		station.xCycleEnable:=FALSE;	
		station.xDone:=TRUE;
		station.xRunningOffProhibit := FALSE ;//运行中信号Off禁止
	1000://XY轴回参考点
				fbXAxisMove.xMoveAuto[1]:=TRUE;
				fbYAxisMove.xMoveAuto[1]:=TRUE;
			IF	fbxAxisMove.xMoveInPos[1] AND 
				fbYAxisMove.xMoveInPos[1] THEN
					station.iStepAuto:= 0;
			END_IF		
{region "清料程序"}
  1010://开始请料
		 //写入数据
			arMainlineFixtureData[arCurFixtureNumStation[5]].xMaterialOnOff:=FALSE;
			arMainlineFixtureData[arCurFixtureNumStation[6]].xMaterialOnOff:=FALSE;
			arMainlineFixtureData[arCurFixtureNumStation[7]].xMaterialOnOff:=FALSE;
			arMainlineFixtureData[arCurFixtureNumStation[8]].xMaterialOnOff:=FALSE;
			arMainlineFixtureData[arCurFixtureNumStation[9]].xMaterialOnOff:=FALSE;		
			arMainlineFixtureData[arCurFixtureNumStation[5]].stProduct.xLidChecking_NOK:=TRUE;
			arMainlineFixtureData[arCurFixtureNumStation[5]].stProduct.xLidChecking_OK:=FALSE;	
			arMainlineFixtureData[arCurFixtureNumStation[6]].stProduct.xLidChecking_NOK:=TRUE;
			arMainlineFixtureData[arCurFixtureNumStation[6]].stProduct.xLidChecking_OK:=FALSE;	
			arMainlineFixtureData[arCurFixtureNumStation[7]].stProduct.xLidChecking_NOK:=TRUE;
			arMainlineFixtureData[arCurFixtureNumStation[7]].stProduct.xLidChecking_OK:=FALSE;	
			arMainlineFixtureData[arCurFixtureNumStation[8]].stProduct.xLidChecking_NOK:=TRUE;
			arMainlineFixtureData[arCurFixtureNumStation[8]].stProduct.xLidChecking_OK:=FALSE;	
			arMainlineFixtureData[arCurFixtureNumStation[9]].stProduct.xLidChecking_NOK:=TRUE;
			arMainlineFixtureData[arCurFixtureNumStation[9]].stProduct.xLidChecking_OK:=FALSE;	
			arMainlineFixtureData[arCurFixtureNumStation[5]].stProduct.xEmptying:=TRUE;
			arMainlineFixtureData[arCurFixtureNumStation[6]].stProduct.xEmptying:=TRUE;
			arMainlineFixtureData[arCurFixtureNumStation[7]].stProduct.xEmptying:=TRUE;
			arMainlineFixtureData[arCurFixtureNumStation[8]].stProduct.xEmptying:=TRUE;
			arMainlineFixtureData[arCurFixtureNumStation[9]].stProduct.xEmptying:=TRUE;		
			station.iStepAuto:=1020;
 1020://XY轴回参考点
				fbXAxisMove.xMoveAuto[1]:=TRUE;
				fbYAxisMove.xMoveAuto[1]:=TRUE;
			IF	fbxAxisMove.xMoveInPos[1] AND 
				fbYAxisMove.xMoveInPos[1] THEN
					station.iStepAuto:= 1100;
			END_IF			
 1100://清料完成
			station.xEmptying:=FALSE;
			station.xEmptyDone:=TRUE;
			station.iStepAuto:=0;
{endregion}			
			
			
			
			
			
		
	ELSE
		;	
END_CASE



END_IF
END_ACTION

ACTION FlowInit:
IF NOT station.xIniting THEN
  station.iStepInit:=0;    
ELSE
//--------------------------------------------初始化步序----------------------------------
CASE station.iStepInit OF	
 0://  
 
  	IF station.xIniting THEN	
  	  station.iStepInit:=10;	
  	END_IF	
10://复位数据
		MEMSET(ADR(arCameraResult),0,SIZEOF(arCameraResult));
		MEMSET(ADR(arCameraResultHmi),0,SIZEOF(arCameraResultHmi));
		FOR i:=2 TO 17 BY 1 DO
			fbCamera[i].xlInit:=TRUE;
			fbCamera[i].xlTrigger:=FALSE;
		END_FOR
		FOR i:=1 TO gc_ModuleProNo BY 1 DO
					MEMSET(ADR(tsModuleProcess[i]),0,SIZEOF(tsModuleProcess[i]));
				END_FOR
		station.iStepInit :=20;
	 
20://伺服上电
  	fbXAxisMove.xPowerInit := TRUE ;
	 fbYAxisMove.xPowerInit := TRUE ;
	 fbZAxisMove.xPowerInit := TRUE ;
	IF fbXAxisMove.xPowerOn AND   fbYAxisMove.xPowerOn AND  fbZAxisMove.xPowerOn THEN 
    	station.iStepInit:=30;	
	END_IF
30://Z轴伺服上升
		fbZAxisMove.xMoveAuto[1]:=TRUE;
		IF fbZAxisMove.xMoveInPos[1]   THEN
			station.iStepInit:=40;	
		END_IF
40://XY轴回参考位置
		fbXAxisMove.xMoveAuto[1]:=TRUE;
		fbYAxisMove.xMoveAuto[1]:=TRUE;
		IF fbXAxisMove.xMoveInPos[1]  AND   fbYAxisMove.xMoveInPos[1]  THEN
			station.iStepInit:=50;	
		END_IF
50://水平调整气缸回原位
				fbHOZAdjustCyl_1.xinit:=TRUE;
        fbHOZAdjustCyl_2.xinit:=TRUE;
        fbHOZAdjustCyl_3.xinit:=true;
       	fbHOZAdjustCyl_4.xinit:=TRUE;
        fbHOZAdjustCyl_5.xinit:=true;
      	fbHOZAdjustCyl_6.xinit:=TRUE;
        fbHOZAdjustCyl_7.xinit:=true;
      	 fbHOZAdjustCyl_8.xinit:=TRUE;
	IF  fbHOZAdjustCyl_1.xHP_Delay AND 
			fbHOZAdjustCyl_2.xHP_Delay AND
			fbHOZAdjustCyl_3.xHP_Delay AND
			fbHOZAdjustCyl_4.xHP_Delay AND 
			fbHOZAdjustCyl_5.xHP_Delay AND 
			fbHOZAdjustCyl_6.xHP_Delay AND
			fbHOZAdjustCyl_7.xHP_Delay AND
			fbHOZAdjustCyl_8.xHP_Delay THEN
		station.iStepInit:=60;	
	END_IF

60://
	station.iStepInit:=100;

100://	
    station.iStepInit:=999;	
999://初始化完成	
	station.iStepInit:=0;
	station.xInitDone:=TRUE;  
END_CASE
END_IF
END_ACTION

ACTION General:
{region "清除过程记录"}
CASE bClearProcessStep OF
	0:	
		IF	 S08_MainLine.xClearProcessStatus THEN
			FOR i:=1 TO gc_ModuleProNo BY 1 DO
				MEMSET(ADR(tsModuleProcess[i]),0,SIZEOF(tsModuleProcess[i]));
			END_FOR
			bClearProcessStep:=10;
		END_IF
	10:
		xClearModuleProcessDone:=TRUE;
		bClearProcessStep:=20;
	20:
		IF NOT S08_MainLine.xClearProcessStatus THEN
			xClearModuleProcessDone:=FALSE;
			bClearProcessStep:=30;
		END_IF
	30:  
			bClearProcessStep:=0;
	
END_CASE
{endregion}

{region "HMI中操作bCounter计数"}
IF station.xSingleRunning THEN
bCounter:=bS03Counter;
END_IF
{endregion}
END_ACTION

ACTION ILC:

//---------------------------------------------------工站可执行-------------------------------------------------------
station.xCanRun :=TRUE ;

//---------------------------------------------------气缸动作条件-------------------------------------------
fbHOZAdjustCyl_1.xOffILC	:=	TRUE	;
fbHOZAdjustCyl_1.xOnILC	:=	TRUE	;
fbHOZAdjustCyl_2.xOffILC	:=	TRUE	;
fbHOZAdjustCyl_2.xOnILC	:=	TRUE	;
fbHOZAdjustCyl_3.xOffILC	:=	TRUE	;
fbHOZAdjustCyl_3.xOnILC	:=	TRUE	;
fbHOZAdjustCyl_4.xOffILC	:=	TRUE	;
fbHOZAdjustCyl_4.xOnILC	:=	TRUE	;
fbHOZAdjustCyl_5.xOffILC	:=	TRUE	;
fbHOZAdjustCyl_5.xOnILC	:=	TRUE	;
fbHOZAdjustCyl_6.xOffILC	:=	TRUE	;
fbHOZAdjustCyl_6.xOnILC	:=	TRUE	;
fbHOZAdjustCyl_7.xOffILC	:=	TRUE	;
fbHOZAdjustCyl_7.xOnILC	:=	TRUE	;
fbHOZAdjustCyl_8.xOffILC	:=	TRUE	;
fbHOZAdjustCyl_8.xOnILC	:=	TRUE	;


//---------------------------------------------------伺服动作条件-------------------------------------------

fbXAxisMove.xRunILC := 		
fbXAxisMove.xMoveILC[1] :=		
fbxAxisMove.xMoveILC[2] :=		
fbxAxisMove.xMoveILC[3] :=		
fbxAxisMove.xMoveILC[4] :=		
fbxAxisMove.xMoveILC[5] := 		TRUE ;//fbZAxisMove.xMoveInPos[1] OR fbZAxisMove.xMoveInPos[2] ;
fbYAxisMove.xRunILC := 		
fbYAxisMove.xMoveILC[1] :=		
fbYAxisMove.xMoveILC[2] :=		
fbYAxisMove.xMoveILC[3] :=		
fbYAxisMove.xMoveILC[4] :=		
fbYAxisMove.xMoveILC[5] := 	TRUE ;//	fbZAxisMove.xMoveInPos[1] OR fbZAxisMove.xMoveInPos[2] ;
fbZAxisMove.xRunILC := 		
fbZAxisMove.xMoveILC[1] :=		
fbZAxisMove.xMoveILC[2] :=		
fbZAxisMove.xMoveILC[3] :=		
fbZAxisMove.xMoveILC[4] :=		
fbZAxisMove.xMoveILC[5] := 		TRUE;

//相机
IF  station.xSingleRunning THEN 
	 FOR  i:=2 TO 17 BY 1 DO
			fbCamera[i].xIDeviceRunning:=TRUE;
	 END_FOR
 ELSE
	 FOR  i:=2 TO 17 BY 1 DO
			fbCamera[i].xIDeviceRunning:=FALSE;
	 END_FOR
END_IF
END_ACTION

ACTION TipAuto:

//------------------------------------------------AutoTip Cylinder--------------------------------
station.adwAutoTip[1].00	:=	fbHOZAdjustCyl_1.xAutoTip	;
//station.adwAutoTip[1].01	:=	fbHOZAdjustCyl_2.xAutoTip	;
station.adwAutoTip[1].02	:=	fbHOZAdjustCyl_3.xAutoTip	;
//station.adwAutoTip[1].03	:=	fbHOZAdjustCyl_4.xAutoTip	;
station.adwAutoTip[1].04	:=	fbHOZAdjustCyl_5.xAutoTip	;
//station.adwAutoTip[1].05	:=	fbHOZAdjustCyl_6.xAutoTip	;
station.adwAutoTip[1].06	:=	fbHOZAdjustCyl_7.xAutoTip	;
//station.adwAutoTip[1].07	:=	fbHOZAdjustCyl_8.xAutoTip	;

//------------------------------------------------AutoTip Servo--------------------------------
//**************************************
FOR i:= 1 TO 5 BY 1 DO 
	IF fbXAxisMove.xMoveAuto[i] THEN
		fbXAxisMove.iPosNumber := i ;
	END_IF
	IF fbYAxisMove.xMoveAuto[i] THEN
		fbYAxisMove.iPosNumber := i ;
	END_IF
	IF fbZAxisMove.xMoveAuto[i] THEN
		fbZAxisMove.iPosNumber := i ;
	END_IF
END_FOR
IF  fbMachine[1].xAutoMode AND NOT fbMachine[1].xRunning  AND arTonDelay[08].Q  THEN
		IF fbXAxisMove.iPosNumber=1 AND NOT fbXAxisMove.xMoveInPos[1] THEN station.adwAutoTip[1].10:=TRUE; END_IF//轴伺服自动时位置不在位置1	
		IF fbXAxisMove.iPosNumber=2 AND NOT fbXAxisMove.xMoveInPos[2] THEN station.adwAutoTip[1].11:=TRUE; END_IF//轴伺服自动时位置不在位置2	
		IF fbXAxisMove.iPosNumber=3 AND NOT fbXAxisMove.xMoveInPos[3] THEN station.adwAutoTip[1].12:=TRUE; END_IF//轴伺服自动时位置不在位置3	
		IF fbXAxisMove.iPosNumber=4 AND NOT fbXAxisMove.xMoveInPos[4] THEN station.adwAutoTip[1].13:=TRUE; END_IF//轴伺服自动时位置不在位置4	
		IF fbXAxisMove.iPosNumber=5 AND NOT fbXAxisMove.xMoveInPos[5] THEN station.adwAutoTip[1].14:=TRUE; END_IF//轴伺服自动时位置不在位置5	
END_IF 		
IF  fbMachine[1].xAutoMode AND NOT fbMachine[1].xRunning  AND arTonDelay[09].Q  THEN		
		IF fbYAxisMove.iPosNumber=1 AND NOT fbYAxisMove.xMoveInPos[1] THEN station.adwAutoTip[1].15:=TRUE; END_IF//轴伺服自动时位置不在位置1	
		IF fbYAxisMove.iPosNumber=2 AND NOT fbYAxisMove.xMoveInPos[2] THEN station.adwAutoTip[1].16:=TRUE; END_IF//轴伺服自动时位置不在位置2	
		IF fbYAxisMove.iPosNumber=3 AND NOT fbYAxisMove.xMoveInPos[3] THEN station.adwAutoTip[1].17:=TRUE; END_IF//轴伺服自动时位置不在位置3	
		IF fbYAxisMove.iPosNumber=4 AND NOT fbYAxisMove.xMoveInPos[4] THEN station.adwAutoTip[1].18:=TRUE; END_IF//轴伺服自动时位置不在位置4	
		IF fbYAxisMove.iPosNumber=5 AND NOT fbYAxisMove.xMoveInPos[5] THEN station.adwAutoTip[1].19:=TRUE; END_IF//轴伺服自动时位置不在位置5	
END_IF 
IF  fbMachine[1].xAutoMode AND NOT fbMachine[1].xRunning  AND arTonDelay[10].Q  THEN		
		IF fbZAxisMove.iPosNumber=1 AND NOT fbZAxisMove.xMoveInPos[1] THEN station.adwAutoTip[1].20:=TRUE; END_IF//轴伺服自动时位置不在位置1	
		IF fbZAxisMove.iPosNumber=2 AND NOT fbZAxisMove.xMoveInPos[2] THEN station.adwAutoTip[1].21:=TRUE; END_IF//轴伺服自动时位置不在位置2	
		IF fbZAxisMove.iPosNumber=3 AND NOT fbZAxisMove.xMoveInPos[3] THEN station.adwAutoTip[1].22:=TRUE; END_IF//轴伺服自动时位置不在位置3	
		IF fbZAxisMove.iPosNumber=4 AND NOT fbZAxisMove.xMoveInPos[4] THEN station.adwAutoTip[1].23:=TRUE; END_IF//轴伺服自动时位置不在位置4	
		IF fbZAxisMove.iPosNumber=5 AND NOT fbZAxisMove.xMoveInPos[5] THEN station.adwAutoTip[1].24:=TRUE; END_IF//轴伺服自动时位置不在位置5			
END_IF
END_ACTION

ACTION TipManual:
//--------------------------------------------ManualTip------------------------------------------------------

//-------------------------------------------气缸提示---------------------------------------------------------




/////////////////////////////////////////////////////////////////////////////////////////////////////////////////
END_ACTION

ACTION Z_Output:
(**************************气缸输出********************************)
//S03上层水平调整气缸1(小)
QxS03HOZAdjustCyl_1WP	:=	fbHOZAdjustCyl_1.xWP_Valve	;
QxS03HOZAdjustCyl_1HP	:=	fbHOZAdjustCyl_1.xHP_Valve	;

QxS03HOZAdjustCyl_2WP	:=	fbHOZAdjustCyl_2.xWP_Valve	;
QxS03HOZAdjustCyl_2HP	:=	fbHOZAdjustCyl_2.xHP_Valve	;

//S03下层水平调整气缸1(小)
QxS03HOZAdjustCyl_3WP	:=	fbHOZAdjustCyl_3.xWP_Valve	;
QxS03HOZAdjustCyl_3HP	:=	fbHOZAdjustCyl_3.xHP_Valve	;

QxS03HOZAdjustCyl_4WP	:=	fbHOZAdjustCyl_4.xWP_Valve	;
QxS03HOZAdjustCyl_4HP	:=	fbHOZAdjustCyl_4.xHP_Valve	;
//S03上层水平调整气缸1(大）
QxS03HOZAdjustCyl_5WP	:=	fbHOZAdjustCyl_5.xWP_Valve	;
QxS03HOZAdjustCyl_5HP	:=	fbHOZAdjustCyl_5.xHP_Valve	;

QxS03HOZAdjustCyl_6WP	:=	fbHOZAdjustCyl_6.xWP_Valve	;
QxS03HOZAdjustCyl_6HP	:=	fbHOZAdjustCyl_6.xHP_Valve	;
//S03下层水平调整气缸1(大）
QxS03HOZAdjustCyl_7WP	:=	fbHOZAdjustCyl_7.xWP_Valve	;
QxS03HOZAdjustCyl_7HP	:=	fbHOZAdjustCyl_7.xHP_Valve	;

QxS03HOZAdjustCyl_8WP	:=	fbHOZAdjustCyl_8.xWP_Valve	;
QxS03HOZAdjustCyl_8HP	:=	fbHOZAdjustCyl_8.xHP_Valve	;
END_ACTION

END_PROGRAM

// ---- POUs/001_Station/S04_AluCovering.TcPOU
PROGRAM S04_AluCovering
VAR
	//工站
	station					: REFERENCE TO FB_Station:=fbstation[4];
	//气缸
	fbHOZAdjustCyl_1	:REFERENCE TO FB_Cylinder:=fbCylinder[20];	//	上层水平调整气缸1
//	fbHOZAdjustCyl_2	:REFERENCE TO FB_Cylinder:=fbCylinder[21];	//	上层水平调整气缸2
	fbHOZAdjustCyl_3	:REFERENCE TO FB_Cylinder:=fbCylinder[22];	//	下层水平调整气缸1
//	fbHOZAdjustCyl_4	:REFERENCE TO FB_Cylinder:=fbCylinder[23];	//	下层水平调整气缸2
	fbAluCoverCyl			:REFERENCE TO FB_Cylinder:=fbCylinder[44];//铝膜胀气轴
	//伺服
	fbZAxisMove_1	 :REFERENCE TO FB_Axis:=fbAxis[10];	//	热熔工位-Z轴伺服1（右）
	fbZAxisMove_2	 :REFERENCE TO FB_Axis:=fbAxis[11];	//		热熔工位-Z轴伺服2
	//温控器
	fbThermostat_1			 :REFERENCE TO FB_TempControl_FUSHI:=fbTempretureControl[1];//温控器1
  fbThermostat_2			 :REFERENCE TO FB_TempControl_FUSHI:=fbTempretureControl[2];//温控器2
	//延时
	arTonDelay :ARRAY[1..20] OF TON;
	//返回值
	UdiReturnValue :ARRAY[1..20] OF UDINT;
	//本地过程数据
	arProcessDataStation : ARRAY [1..2] OF DUT_MainlineFixture;
	i: INT;
	//过程记录
	tsModuleProcess:ARRAY[1..gc_ModuleProNo] OF DUT_Process;
	xClearModuleProcessDone:BOOL;
	bClearProcessStep	:BYTE;
END_VAR

A_Input();
Alarm();
Delay();
FlowAuto();
FlowInit();
General();
ILC();
TipAuto();
TipManual();
Z_Output();

ACTION A_Input:
//气缸
fbHOZAdjustCyl_1.xWP_Sensor	:=	IxS04HOZAdjustCyl_1WP AND IxS04HOZAdjustCyl_2WP	;
fbHOZAdjustCyl_1.xHP_Sensor	:=	IxS04HOZAdjustCyl_1HP	 AND IxS04HOZAdjustCyl_2hP;
fbHOZAdjustCyl_3.xWP_Sensor	:=	IxS04HOZAdjustCyl_3WP	 AND IxS04HOZAdjustCyl_4WP;
fbHOZAdjustCyl_3.xHP_Sensor	:=	IxS04HOZAdjustCyl_3HP	AND IxS04HOZAdjustCyl_4HP;

fbAluCoverCyl.xWP_Sensor :=fbAluCoverCyl.xWP_Valve;
fbAluCoverCyl.xHP_Sensor:=fbAluCoverCyl.xHP_Valve;
END_ACTION

ACTION Alarm:
station.adwAlarm[1].00	:=	station.xInitTimeout	;//	S04 初始化超时
station.adwAlarm[1].01	:=	fbHOZAdjustCyl_1.xHP_Off 	;//	S04上层水平调整气缸1原点未到位
station.adwAlarm[1].02	:=	fbHOZAdjustCyl_1.xWP_Off 	;//	S04上层水平调整气缸1动点未到位
station.adwAlarm[1].03	:=	fbHOZAdjustCyl_3.xHP_Off	;//	S04下层水平调整气缸1原点未到位
station.adwAlarm[1].04	:=	fbHOZAdjustCyl_3.xWP_Off	;//	S04下层水平调整气缸1动点未到位
station.adwAlarm[1].05	:=	fbZAxisMove_1.xError	;//	S04热封铝膜工位Z轴伺服1报错
station.adwAlarm[1].06	:=	fbZAxisMove_1.xNotPowerOn	;//	S04热封铝膜工位Z轴伺服1未使能
station.adwAlarm[1].07	:=	fbZAxisMove_1.xMoveTimeout	;//	S04热封铝膜工位Z轴伺服1移动超时
station.adwAlarm[1].08	:=	fbZAxisMove_2.xError	;//	S04热封铝膜工位Z轴伺服2报错
station.adwAlarm[1].09	:=	fbZAxisMove_2.xNotPowerOn	;//	S04热封铝膜工位Z轴伺服2未使能
station.adwAlarm[1].10	:=	fbZAxisMove_2.xMoveTimeout	;//	S04热封铝膜工位Z轴伺服2移动超时
station.adwAlarm[1].11	:=	fbThermostat_1.xError	;//	S04热封铝膜工位温控器1报错
station.adwAlarm[1].12	:=	fbThermostat_2.xError	;//	S04热封铝膜工位温控器2报错
END_ACTION

ACTION Delay:
arTonDelay[01](IN:= , PT:=T#0.1S , Q=> , ET=> );
arTonDelay[02](IN:=  , PT:=stData.Thermostat[1].tTON_Delay , Q=> , ET=> );//热熔延时时间
arTonDelay[03](IN:=   , PT:=T#1S , Q=> , ET=> );
arTonDelay[04](IN:= , PT:=T#0.1S , Q=> , ET=> );
arTonDelay[05](IN:= , PT:=T#0.1S , Q=> , ET=> );
arTonDelay[06](IN:= , PT:=T#0.1S , Q=> , ET=> );
arTonDelay[07](IN:= , PT:=T#0.1S , Q=> , ET=> );
arTonDelay[08](IN:= , PT:=T#0.1S , Q=> , ET=> );
arTonDelay[09](IN:= NOT fbZAxisMove_1.xbusy, PT:=T#0.1S , Q=> , ET=> );//TipAuto使用
arTonDelay[10](IN:= NOT fbZAxisMove_2.xbusy, PT:=T#0.1S , Q=> , ET=> );//TipAuto使用
END_ACTION

ACTION FlowAuto:

//-----------------------------------------初始化是否完成判断----------------------------------------------
IF NOT station.xInitDone 
THEN
 	station.iStepAuto:=0;
 	station.xDone:=FALSE;
	station.xRunningOffProhibit := FALSE ;//运行中信号Off禁止
ELSIF station.xRunning  OR (  tsModuleProcess[2].xProcessStarted AND   NOT tsModuleProcess[2].xProcessCompleted)//Z轴热熔
THEN
//-----------------------------------------动作步骤--------------------------------------------------------
CASE station.iStepAuto OF	  
	0: //----Home Step，等待启动----
		IF station.xDisabled 
			AND station.xCanRun 
			AND NOT fbMachine[1].xStopped 
			AND NOT station.xSingleRunning 
		THEN
			station.xDone:=TRUE;
		END_IF
		
		IF  station.xSingleRunning 
			OR station.xCanRun 
			AND NOT station.xDone 
			AND NOT station.xDisabled 
			AND NOT fbMachine[1].xStopped
		THEN
			station.xCycleEnable:=TRUE;
			station.xDone:= FALSE;  
			station.xRunningOffProhibit := TRUE ;//运行中信号Off禁止
			station.iStepAuto:= 10;
		END_IF
    10: //复位数据
			(*开启控温系统*) 
			fbThermostat_1.xStart :=TRUE;
			fbThermostat_2.xStart :=TRUE;
			arTonDelay[02](IN:= FALSE);
				 FOR i:=1 TO gc_ModuleProNo BY 1 DO
						 MEMSET(ADR(tsModuleProcess[i]),0,SIZEOF(tsModuleProcess[i]));
				 END_FOR
			station.iStepAuto:=20;	
	20:////Restore_after_Estop_Process1 上载数据流程
			IF  station.xSingleRunning THEN // OR  fbMachine[1].xTryRun THEN
					station.iStepAuto:=50;
			ELSIF tsModuleProcess[1].xProcessNotStarted AND NOT  tsModuleProcess[1].xProcessStarted THEN
					station.iStepAuto :=21; (*process not started*)
			ELSIF  tsModuleProcess[1].xProcessStarted AND NOT  tsModuleProcess[1].xProcessCompleted THEN
				 station.iStepAuto := 21;(*process started*)
			ELSIF  tsModuleProcess[1].xProcessCompleted AND NOT tsModuleProcess[1].xQDataCompleted  THEN
					station.iStepAuto := 40 ;(*process completed*)
			ELSIF tsModuleProcess[1].xQDataCompleted THEN
					station.iStepAuto :=40;(*Qdata completed *)
			ELSE
					station.iStepAuto :=21; 
			END_IF	
	21://
				tsModuleProcess[1].xProcessNotStarted:=TRUE;
				station.iStepAuto:= 30;
				
	30://数据load 
			 tsModuleProcess[1].xProcessStarted	:=TRUE;
			 MEMCPY(ADR(arProcessDataStation[1]),ADR(arMainlineFixtureData[arCurFixtureNumStation[10]]),SIZEOF(arMainlineFixtureData[arCurFixtureNumStation[10]]));
			 MEMCPY(ADR(arProcessDataStation[2]),ADR(arMainlineFixtureData[arCurFixtureNumStation[11]]),SIZEOF(arMainlineFixtureData[arCurFixtureNumStation[11]]));
			 tsModuleProcess[1].xProcessCompleted:=TRUE;
			 tsModuleProcess[1].xQDataCompleted:=TRUE;
			 station.iStepAuto:= 40;
	40: //判断产品状态
			IF	NOT fbMachine[1].xTryRun THEN
						 IF  station.xEmptyDone THEN
											 station.iStepAuto:= 999;	
						 ELSIF  arProcessDataStation[1].stProduct.xEmptying  AND 
										arProcessDataStation[2].stProduct.xEmptying  THEN
											 station.xEmptying:=TRUE;
											 station.iStepAuto:= 1000;
						 ELSIF  arProcessDataStation[1].xMaterialOnOff   AND
										arProcessDataStation[2].xMaterialOnOff  THEN
											 station.iStepAuto:= 41;
						 ELSIF	 NOT arProcessDataStation[1].xMaterialOnOff   AND
										NOT arProcessDataStation[2].xMaterialOnOff  THEN
											 station.iStepAuto:= 999;
						 END_IF
			ELSE
						station.iStepAuto:= 41;
			END_IF
	41://手动NOK按钮
			IF   arManualNOKHmiButton[4]  AND NOT station.xCycleRunning THEN
				station.iStepAuto:= 140;
			ELSE	
				station.iStepAuto:= 50;
			END_IF	
	
	/////产品流程开始	
	50:////Restore_after_Estop_Process2 热熔流程
			IF  station.xSingleRunning OR fbMachine[1].xTryRun THEN
					station.iStepAuto :=60; 
			ELSIF tsModuleProcess[2].xProcessNotStarted AND NOT  tsModuleProcess[2].xProcessStarted THEN
					station.iStepAuto :=60; (*process not started*)
			ELSIF  tsModuleProcess[2].xProcessStarted AND NOT  tsModuleProcess[2].xProcessCompleted THEN
				 station.iStepAuto := 140;(*process started*)
			ELSIF  tsModuleProcess[2].xProcessCompleted AND NOT tsModuleProcess[2].xQDataCompleted  THEN
					station.iStepAuto :=130;(*process completed*)
			ELSIF tsModuleProcess[2].xQDataCompleted THEN
					station.iStepAuto :=160;(*Qdata completed *)
			ELSE
					station.iStepAuto :=60; 
			END_IF	
	60://
				 tsModuleProcess[2].xProcessNotStarted:=TRUE;
				 station.iStepAuto :=70; 
	70://水平调整气缸伸出
					IF  iBoxChoose =1 THEN
						(*上层水平调整气缸*)
						fbHOZAdjustCyl_1.xAuto :=TRUE;
					//	fbHOZAdjustCyl_2.xAuto :=TRUE;
						IF  fbHOZAdjustCyl_1.xWP_Delay  THEN // AND fbHOZAdjustCyl_2.xWP_Delay  THEN
								station.iStepAuto:= 80;
						END_IF
					ELSIF  iBoxChoose= 2 THEN
						(*下层水平调整气缸*)
						fbHOZAdjustCyl_3.xAuto :=TRUE;
					//	fbHOZAdjustCyl_4.xAuto :=TRUE;
						IF  fbHOZAdjustCyl_3.xWP_Delay  THEN  //AND fbHOZAdjustCyl_4.xWP_Delay  THEN
								station.iStepAuto:= 80;
						END_IF
					END_IF
	
	80://判断加热棒是否准备就绪
			IF  ( fbThermostat_1.xRdy AND  fbThermostat_2.xRdy ) OR 
				axBypassSignal[4] OR  fbMachine[1].xTryRun THEN
					station.iStepAuto:= 90;
			END_IF
	90://Z轴伺服下降到位置1
			tsModuleProcess[2].xProcessStarted:=TRUE;
			fbZAxisMove_1.xMoveAuto[2]:=TRUE;
			fbZAxisMove_2.xMoveAuto[2]:=TRUE;
			IF  fbZAxisMove_1.xMoveInPos[2] AND fbZAxisMove_2.xMoveInPos[2]THEN
				station.iStepAuto:=100;	
			END_IF
	100://复位热熔时间
			arTonDelay[02](IN:=FALSE  , PT:=stData.Thermostat[1].tTON_Delay , Q=> , ET=> );//热熔延时时间
			station.iStepAuto:=110;
 	110://延时等待热熔完成
			arTonDelay[02](IN:=TRUE  , PT:=stData.Thermostat[1].tTON_Delay , Q=> , ET=> );//热熔延时时间
		IF  arTonDelay[02].Q  OR axBypassSignal[4]  OR fbMachine[1].xTryRun  THEN
			station.iStepAuto:=120;	
			arTonDelay[02](IN:= FALSE );//热熔延时时间
		END_IF
	120://
			
			station.iStepAuto:=130;	
	130://结果OK
			arProcessDataStation[1].stProduct.xAluCovering_NOK:=FALSE;
			arProcessDataStation[1].stProduct.xAluCovering_OK:=TRUE;
			arProcessDataStation[2].stProduct.xAluCovering_NOK:=FALSE;
			arProcessDataStation[2].stProduct.xAluCovering_OK:=TRUE;
			station.iStepAuto:=150;	
	140://结果NG 
			arProcessDataStation[1].stProduct.xAluCovering_NOK:=TRUE;
			arProcessDataStation[1].stProduct.xAluCovering_OK:=FALSE;
			arProcessDataStation[2].stProduct.xAluCovering_NOK:=TRUE;
			arProcessDataStation[2].stProduct.xAluCovering_OK:=FALSE;
			station.iStepAuto:=150;	
	150:
			tsModuleProcess[2].xQDataCompleted :=TRUE;
			station.iStepAuto:=160;	
	160://Z轴上升
			fbZAxisMove_1.xMoveAuto[1]:=TRUE;
			fbZAxisMove_2.xMoveAuto[1]:=TRUE;
			IF  fbZAxisMove_1.xMoveInPos[1] AND fbZAxisMove_2.xMoveInPos[1]THEN
				station.iStepAuto:=170;	
			END_IF
	170://水平调整气缸收回
			tsModuleProcess[2].xProcessCompleted :=TRUE;
			fbHOZAdjustCyl_1.xAuto :=FALSE;
		//	fbHOZAdjustCyl_2.xAuto :=false;
			fbHOZAdjustCyl_3.xAuto :=false;
		//	fbHOZAdjustCyl_4.xAuto :=false;
		IF	fbHOZAdjustCyl_1.xhp_Delay AND
		 //   fbHOZAdjustCyl_2.xhp_Delay and
		    fbHOZAdjustCyl_3.xhp_Delay  THEN
		 //   fbHOZAdjustCyl_4.xhp_Delay THEN
			station.iStepAuto:=200;	
		END_IF
	////产品流程结束	
	200:////Restore_after_Estop_Process3 数据传输流程
			IF  station.xSingleRunning THEN //OR fbMachine[1].xTryRun THEN
					station.iStepAuto :=999; 
			ELSIF tsModuleProcess[3].xProcessNotStarted AND NOT  tsModuleProcess[3].xProcessStarted THEN
					station.iStepAuto :=210; (*process not started*)
			ELSIF  tsModuleProcess[3].xProcessStarted AND NOT  tsModuleProcess[3].xProcessCompleted THEN
				 station.iStepAuto := 220;(*process started*)
			ELSIF  tsModuleProcess[3].xProcessCompleted AND NOT tsModuleProcess[3].xQDataCompleted  THEN
					station.iStepAuto :=230;(*process completed*)
			ELSIF tsModuleProcess[3].xQDataCompleted THEN
					station.iStepAuto :=999;(*Qdata completed *)
			ELSE
					station.iStepAuto :=210; 
			END_IF		
	210://		
				tsModuleProcess[3].xProcessNotStarted:=TRUE;
				station.iStepAuto :=220; 
	220://数据unload
		tsModuleProcess[3].xProcessStarted:=TRUE;
		MEMCPY(ADR(arMainlineFixtureData[arCurFixtureNumStation[10]]),ADR(arProcessDataStation[1]),SIZEOF(arProcessDataStation[1]));
		MEMCPY(ADR(arMainlineFixtureData[arCurFixtureNumStation[11]]),ADR(arProcessDataStation[2]),SIZEOF(arProcessDataStation[2]));
		station.iStepAuto:= 230;
	230://
			tsModuleProcess[3].xProcessCompleted:=TRUE;
			station.iStepAuto :=240; 
 	240://本地数据清除
		//	MEMSET(ADR(arProcessDataStation[1]),0,SIZEOF(arProcessDataStation[1]));
		//	MEMSET(ADR(arProcessDataStation[2]),0,SIZEOF(arProcessDataStation[2]));
			arManualNOKHmiButton[4]:=FALSE;
			tsModuleProcess[3].xQDataCompleted:=TRUE;
			station.iStepAuto:= 999;
	999://----Single Run Finish----
		station.iStepAuto :=0;
		IF NOT station.xSingleContinuousRun THEN
			station.xSingleRunFlag:=FALSE;
		END_IF
		station.xCycleEnable:=FALSE;	
		station.xDone:=TRUE;
	
{region "清料程序"}
1000://写入数据
	 		arProcessDataStation[1].xMaterialOnOff:=FALSE;
			arProcessDataStation[2].xMaterialOnOff:=FALSE;
	 		arProcessDataStation[1].stProduct.xAluCovering_NOK:=FALSE;
			arProcessDataStation[2].stProduct.xAluCovering_OK:=FALSE;
			arProcessDataStation[1].stProduct.xAluCovering_NOK:=FALSE;
			arProcessDataStation[2].stProduct.xAluCovering_OK:=FALSE;
			arProcessDataStation[1].stProduct.xEmptying:=TRUE;
			arProcessDataStation[2].stProduct.xEmptying:=TRUE;
			MEMCPY(ADR(arMainlineFixtureData[arCurFixtureNumStation[10]]),ADR(arProcessDataStation[1]),SIZEOF(arProcessDataStation[1]));
			MEMCPY(ADR(arMainlineFixtureData[arCurFixtureNumStation[11]]),ADR(arProcessDataStation[2]),SIZEOF(arProcessDataStation[2]));
			station.iStepAuto:= 1010;
1010://Z轴回参考位置
			fbZAxisMove_1.xMoveAuto[1]:=TRUE;
			fbZAxisMove_2.xMoveAuto[1]:=TRUE;
			IF  fbZAxisMove_1.xMoveInPos[1] AND fbZAxisMove_2.xMoveInPos[1]THEN
				station.iStepAuto:=1020;	
			END_IF	 
1020://清料完成
	 		station.xEmptying:=FALSE;
		  station.xEmptyDone:=TRUE;
			station.iStepAuto:=0;
{endRegion}	
		
		
		
		
		
		
		
		
		
		
		
		
		
	ELSE
		;	
END_CASE



END_IF
END_ACTION

ACTION FlowInit:
IF NOT station.xIniting THEN
  station.iStepInit:=0;    
ELSE
//--------------------------------------------初始化步序----------------------------------
CASE station.iStepInit OF	
 0://  
  	IF station.xIniting THEN	
  	  station.iStepInit:=10;	
  	END_IF	
10://复位数据
		FOR i:=1 TO gc_ModuleProNo BY 1 DO
				MEMSET(ADR(tsModuleProcess[i]),0,SIZEOF(tsModuleProcess[i]));
			END_FOR
	 station.iStepInit:=20;	
20://关闭控温系统
	fbThermostat_1.xStart :=FALSE;
	fbThermostat_2.xStart :=FALSE;
	 station.iStepInit:=30;	
30://Z轴伺服上电
	fbZAxisMove_1.xPowerInit:=TRUE;
    fbZAxisMove_2.xPowerInit:=TRUE;
	IF  fbZAxisMove_1.xPowerOn AND fbZAxisMove_2.xPowerOn THEN
		station.iStepInit:=40;	
	END_IF
40://Z轴伺服上升
	fbZAxisMove_1.xMoveAuto[1]:=TRUE;
    fbZAxisMove_2.xMoveAuto[1]:=TRUE;
	IF  fbZAxisMove_1.xMoveInPos[1] AND fbZAxisMove_2.xMoveInPos[1]THEN
		station.iStepInit:=50;	
	END_IF
50://水平调整气缸收回
	fbHOZAdjustCyl_1.xinit:=TRUE;	
//	fbHOZAdjustCyl_2.xinit:=true;	
	fbHOZAdjustCyl_3.xinit:=true;	
//	fbHOZAdjustCyl_4.xinit:=true;		
	IF     fbHOZAdjustCyl_1.xHp_Delay  AND 
	//	   fbHOZAdjustCyl_2.xHp_Delay  AND 
	 	   fbHOZAdjustCyl_3.xHp_Delay  THEN 
    //       fbHOZAdjustCyl_4.xHp_Delay  THEN
			station.iStepInit:=100;
	END_IF
100://	
    station.iStepInit:=999;	
999://初始化完成	
	station.iStepInit:=0;
	station.xInitDone:=TRUE;  
END_CASE
END_IF
END_ACTION

ACTION General:
(******************清除过程记录**********************)
CASE bClearProcessStep OF
	0:	
		IF	 S08_MainLine.xClearProcessStatus THEN
			FOR i:=1 TO gc_ModuleProNo BY 1 DO
				MEMSET(ADR(tsModuleProcess[i]),0,SIZEOF(tsModuleProcess[i]));
			END_FOR
			bClearProcessStep:=10;
		END_IF
	10:
		xClearModuleProcessDone:=TRUE;
		bClearProcessStep:=20;
	20:
		IF NOT S08_MainLine.xClearProcessStatus THEN
			xClearModuleProcessDone:=FALSE;
			bClearProcessStep:=30;
		END_IF
	30:  
			bClearProcessStep:=0;
	
END_CASE
END_ACTION

ACTION ILC:

//---------------------------------------------------工站可执行-------------------------------------------------------
station.xCanRun :=TRUE ;

//---------------------------------------------------气缸动作条件-------------------------------------------
fbHOZAdjustCyl_1.xOffILC	:=	TRUE	;
fbHOZAdjustCyl_1.xOnILC	:=	TRUE	;
//fbHOZAdjustCyl_2.xOffILC	:=	TRUE	;
//fbHOZAdjustCyl_2.xOnILC	:=	TRUE	;
fbHOZAdjustCyl_3.xOffILC	:=	TRUE	;
fbHOZAdjustCyl_3.xOnILC	:=	TRUE	;
//fbHOZAdjustCyl_4.xOffILC	:=	TRUE	;
//fbHOZAdjustCyl_4.xOnILC	:=	TRUE	;


//---------------------------------------------------伺服动作条件-------------------------------------------

fbZAxisMove_1.xRunILC := 
fbZAxisMove_1.xMoveILC[1] :=
fbZAxisMove_1.xMoveILC[2] :=
fbZAxisMove_1.xMoveILC[3] :=
fbZAxisMove_1.xMoveILC[4] :=
fbZAxisMove_1.xMoveILC[5] := TRUE ;

fbZAxisMove_2.xRunILC := 
fbZAxisMove_2.xMoveILC[1] :=
fbZAxisMove_2.xMoveILC[2] :=
fbZAxisMove_2.xMoveILC[3] :=
fbZAxisMove_2.xMoveILC[4] :=
fbZAxisMove_2.xMoveILC[5] := TRUE ;

fbAluCoverCyl.xOffILC:=true;
fbAluCoverCyl.xOnILC:=true;
END_ACTION

ACTION TipAuto:

//------------------------------------------------AutoTip Cylinder--------------------------------
station.adwAutoTip[1].00	:=	fbHOZAdjustCyl_1.xAutoTip	;
//station.adwAutoTip[1].01	:=	fbHOZAdjustCyl_2.xAutoTip	;
station.adwAutoTip[1].02	:=	fbHOZAdjustCyl_3.xAutoTip	;
//station.adwAutoTip[1].03	:=	fbHOZAdjustCyl_4.xAutoTip	;
	
//------------------------------------------------AutoTip Servo--------------------------------
//**************************************
FOR i:= 1 TO 5 BY 1 DO 
	IF fbZAxisMove_1.xMoveAuto[i] THEN
		fbZAxisMove_1.iPosNumber := i ;
	END_IF
	IF fbZAxisMove_2.xMoveAuto[i] THEN
		fbZAxisMove_2.iPosNumber := i ;
	END_IF
	
END_FOR

IF  fbMachine[1].xAutoMode AND NOT fbMachine[1].xRunning AND arTonDelay[9].Q  THEN
	IF	fbZAxisMove_1.iPosNumber=1 	AND NOT fbZAxisMove_1.xMoveInPos[1] 	THEN 	station.adwAutoTip[1].10:=TRUE	;	END_IF//轴伺服自动时位置不在位置1
	if	fbZAxisMove_1.iPosNumber=2	AND NOT fbZAxisMove_1.xMoveInPos[2]	THEN 	station.adwAutoTip[1].11:=TRUE	;	END_IF//轴伺服自动时位置不在位置2
	if	fbZAxisMove_1.iPosNumber=3	AND NOT fbZAxisMove_1.xMoveInPos[3]	THEN 	station.adwAutoTip[1].12:=TRUE	;	END_IF//轴伺服自动时位置不在位置3
	if	fbZAxisMove_1.iPosNumber=4	AND NOT fbZAxisMove_1.xMoveInPos[4]	THEN 	station.adwAutoTip[1].13:=TRUE	;	END_IF//轴伺服自动时位置不在位置4
	IF	fbZAxisMove_1.iPosNumber=5	AND NOT fbZAxisMove_1.xMoveInPos[5]	THEN 	station.adwAutoTip[1].14:=TRUE	;	END_IF//轴伺服自动时位置不在位置5
END_IF
IF  fbMachine[1].xAutoMode AND NOT fbMachine[1].xRunning AND arTonDelay[10].Q  THEN
	IF	fbZAxisMove_2.iPosNumber=1 	AND NOT fbZAxisMove_2.xMoveInPos[1] 	THEN 	station.adwAutoTip[1].15:=TRUE	;	END_IF//轴伺服自动时位置不在位置1
	if	fbZAxisMove_2.iPosNumber=2	AND NOT fbZAxisMove_2.xMoveInPos[2]	THEN 	station.adwAutoTip[1].16:=TRUE	;	END_IF//轴伺服自动时位置不在位置2
	if	fbZAxisMove_2.iPosNumber=3	AND NOT fbZAxisMove_2.xMoveInPos[3]	THEN 	station.adwAutoTip[1].17:=TRUE	;	END_IF//轴伺服自动时位置不在位置3
	if	fbZAxisMove_2.iPosNumber=4	AND NOT fbZAxisMove_2.xMoveInPos[4]	THEN 	station.adwAutoTip[1].18:=TRUE	;	END_IF//轴伺服自动时位置不在位置4
	if	fbZAxisMove_2.iPosNumber=5	AND NOT fbZAxisMove_2.xMoveInPos[5]	THEN 	station.adwAutoTip[1].19:=TRUE	;	END_IF//轴伺服自动时位置不在位置5
END_IF
END_ACTION

ACTION TipManual:
//--------------------------------------------ManualTip------------------------------------------------------

//-------------------------------------------气缸提示---------------------------------------------------------




/////////////////////////////////////////////////////////////////////////////////////////////////////////////////
END_ACTION

ACTION Z_Output:
(**************************气缸输出********************************)
QxS04HOZAdjustCyl_1WP	:=	fbHOZAdjustCyl_1.xWP_Valve	;
QxS04HOZAdjustCyl_1HP	:=	fbHOZAdjustCyl_1.xHP_Valve	;

QxS04HOZAdjustCyl_3WP	:=	fbHOZAdjustCyl_3.xWP_Valve	;
QxS04HOZAdjustCyl_3HP	:=	fbHOZAdjustCyl_3.xHP_Valve	;

QxS04AluCoverCylWP:=fbAluCoverCyl.xWP_Valve;
END_ACTION

END_PROGRAM

// ---- POUs/003_FB/064_Temperature/FB_TempControl_FUSHI.TcPOU
FUNCTION_BLOCK FB_TempControl_FUSHI
(*
********************************************************************************
* Name: FB_TempControl_FUSHI
*
* Author:  AutomanH
* Version: 1.0.0
*
* Description:
* 
*
* Remarks:
*
* Revisions:
*   V2.0.0 -Automanh 2022.07.01  add Power on singal PWM Countrol for temperature up Lower
********************************************************************************************)
VAR_INPUT
	xEstop		:BOOL;//急停
	xStart		:BOOL;//控温开始
	xSvSet		:BOOL;//温度设置
	stSysPar	:ST_FUSHI_PXF_Sys_Pointer;
	stPar		  :ST_FUSHI_PXF_ParSet;
END_VAR
VAR_OUTPUT
	stParRead	:ST_FUSHI_PXF_ParRead;
	xRdy		:BOOL;//温度就绪
	xPowerOut	:BOOL;//功率输出
	xError		:BOOL;
	sError		:STRING;
END_VAR
VAR
	{attribute 'tc_no_symbol'}	
	_diCmdState:INT;
	{attribute 'tc_no_symbol'}
	_tonDelay,_tonCmdTimeout:TON;
	{attribute 'tc_no_symbol'}
	///ReadStatus
	_aRead_VAR: FB_MBReadInputRegs;
	{attribute 'tc_no_symbol'}
	//Set SV
	_aWtirt_VAR: FB_MBWriteRegs;
	{attribute 'tc_no_symbol'}
  _rSvSet	:R_TRIG;
	{attribute 'tc_no_symbol'}	
	fbTon1:TON;
	{attribute 'tc_no_symbol'}
	tCycleTime:TIME;
END_VAR

ACT_Connect();
M_DutyRatio();
IF stPar.iMaxTemperature=0 THEN
	stPar.iMaxTemperature:=230;	
END_IF
IF stPar.iMinTemperature>stPar.iMaxTemperature THEN
	stPar.iMinTemperature:=0;	
END_IF

IF xEstop THEN
	xPowerOut:=xStart AND stParRead.iPV<stPar.iMaxTemperature AND stParRead.iPV>stPar.iMinTemperature AND (stParRead.iPV-stParRead.iSV<15) ;
ELSE
	xPowerOut:=FALSE;
	xRdy:=FALSE;
END_IF

//温度就绪
xRdy:=(stParRead.iPV>stParRead.iSV-3) AND (stParRead.iPV<=stParRead.iSV+8) AND NOT xError AND xEstop;

//
IF stSysPar.strSlaveIP<>''  THEN
   IF stSysPar.bySlaveID<>0 AND stSysPar.iSlavePort<>0 THEN
      _aRead_VAR.bExecute:=stSysPulse.xP200ms; //温度读取
			IF xSvSet THEN   //温度设置
	      IF xError OR stParRead.iSV=stPar.iSV THEN
		       xSvSet:=FALSE;
	      END_IF
      END_IF
	 END_IF	 
END_IF

_rSvSet(CLK:=xSvSet);
_aWtirt_VAR.bExecute:=_rSvSet.Q; //温度设置

ACTION ACT_Connect:
	_aRead_VAR(
	sIPAddr:= stSysPar.strSlaveIP,
	nTCPPort:= stSysPar.iSlavePort, 
	nUnitID:= stSysPar.bySlaveID, 
	nQuantity:= 5, 
	nMBAddr:= 2000, 
	cbLength:= 10, 
	pDestAddr:= ADR(stParRead), 
	bExecute:= , 
	tTimeout:= T#1S, 
	bBusy=> , 
	bError=> , 
	nErrId=> , 
	cbRead=> );	
 
_aWtirt_VAR(
	sIPAddr:= stSysPar.strSlaveIP, 
	nTCPPort:= stSysPar.iSlavePort, 
	nUnitID:= stSysPar.bySlaveID, 
	nQuantity:=1 , 
	nMBAddr:= 2002, 
	cbLength:=2 , 
	pSrcAddr:= ADR(stPar.iSV), 
	bExecute:= , 
	tTimeout:= , 
	bBusy=> , 
	bError=> , 
	nErrId=> );	
sError:='';

IF _aRead_VAR.nErrId<>0 OR _aWtirt_VAR.nErrId<>0 THEN
	sError:=TO_STRING(_aRead_VAR.nErrId XOR _aWtirt_VAR.nErrId);
ELSIF	stPar.iSV>stPar.iMaxTemperature THEN
	sError:=CONCAT(sError,'设定值超出温度上限');	
ELSIF	stPar.iSV<stPar.iMinTemperature THEN
	sError:=CONCAT(sError,'设定值低于温度下限');
ELSIF	stParRead.iPV>stPar.iMaxTemperature THEN
	sError:=CONCAT(sError,'当前值超出温度上限');	
ELSIF	stParRead.iPV<stPar.iMinTemperature THEN
	sError:=CONCAT(sError,'当前低于温度下限');		
ELSIF	ABS(stParRead.iDV)>10 AND stParRead.iPV>stParRead.iSV THEN
	sError:=CONCAT(sError,'温度超差过大');
ELSIF	ABS(stParRead.iDV)>10 AND stParRead.iPV<stParRead.iSV THEN
	sError:=CONCAT(sError,'温度差距过大');	
END_IF
END_ACTION

METHOD M_DutyRatio : BOOL
fbTon1(IN:= NOT fbTon1.Q, PT:=tCycleTime , Q=> , ET=> );
//33％ on 66％ off
M_DutyRatio:=fbton1.ET>fbton1.PT/3;
END_METHOD

END_FUNCTION_BLOCK

// ---- POUs/001_Station/S05_Adjusting.TcPOU
PROGRAM S05_Adjusting

VAR
	//工站
	station					: REFERENCE TO FB_Station:=fbstation[5];
	//气缸




	//伺服
	fbZAxisMove_1	 :REFERENCE TO FB_Axis:=fbAxis[12];	//	调整工位-Z轴伺服1
	fbZAxisMove_2	 :REFERENCE TO FB_Axis:=fbAxis[13];	//	调整工位-Z轴伺服2



	//延时
	arTonDelay :ARRAY[1..20] OF TON;
	//返回值
	UdiReturnValue :ARRAY[1..20] OF UDINT;
	//本地过程数据
	arProcessDataStation : ARRAY [1..2] OF DUT_MainlineFixture;
	i: INT;
	//过程记录
	tsModuleProcess:ARRAY[1..gc_ModuleProNo] OF DUT_Process;
	xClearModuleProcessDone:BOOL;
	bClearProcessStep	:BYTE;
END_VAR

A_Input();
Alarm();
Delay();
FlowAuto();
FlowInit();
General();
ILC();
TipAuto();
TipManual();
Z_Output();

ACTION A_Input:
//气缸
END_ACTION

ACTION Alarm:
station.adwAlarm[1].00	:=	station.xInitTimeout	;//	S05 初始化超时
station.adwAlarm[1].01	:=	fbZAxisMove_1.xError	;//	S05调整工位Z轴伺服1报错
station.adwAlarm[1].02	:=	fbZAxisMove_1.xNotPowerOn	;//	S05调整工位Z轴伺服1未使能
station.adwAlarm[1].03	:=	fbZAxisMove_1.xMoveTimeout	;//	S05调整工位Z轴伺服1移动超时
station.adwAlarm[1].04	:=	fbZAxisMove_2.xError	;//	S05调整工位Z轴伺服2报错
station.adwAlarm[1].05	:=	fbZAxisMove_2.xNotPowerOn	;//	S05调整工位Z轴伺服2未使能
station.adwAlarm[1].06	:=	fbZAxisMove_2.xMoveTimeout	;//	S05调整工位Z轴伺服2移动超时
END_ACTION

ACTION Delay:
(*arTonDelay[01](IN:= , PT:=T#0.1S , Q=> , ET=> );*)//TipAuto使用
arTonDelay[02](IN:=  , PT:=T#1S , Q=> , ET=> );//伺服下压延时
arTonDelay[03](IN:=   , PT:=T#1S , Q=> , ET=> );
arTonDelay[04](IN:= , PT:=T#0.1S , Q=> , ET=> );
arTonDelay[05](IN:= , PT:=T#0.1S , Q=> , ET=> );
arTonDelay[06](IN:= , PT:=T#0.1S , Q=> , ET=> );
arTonDelay[07](IN:= , PT:=T#0.1S , Q=> , ET=> );
arTonDelay[08](IN:= , PT:=T#0.1S , Q=> , ET=> );
arTonDelay[09](IN:= NOT fbZAxisMove_1.xbusy, PT:=T#0.1S , Q=> , ET=> );//TipAuto使用
arTonDelay[10](IN:= NOT fbZAxisMove_2.xbusy, PT:=T#0.1S , Q=> , ET=> );//TipAuto使用
END_ACTION

ACTION FlowAuto:

//-----------------------------------------初始化是否完成判断----------------------------------------------
IF NOT station.xInitDone 
THEN
 	station.iStepAuto:=0;
 	station.xDone:=FALSE;
ELSIF station.xRunning  OR 
(  tsModuleProcess[2].xProcessStarted AND   NOT tsModuleProcess[2].xProcessCompleted)//Z周调整
THEN
//-----------------------------------------动作步骤--------------------------------------------------------
CASE station.iStepAuto OF	  
	0: //----Home Step，等待启动----
		IF station.xDisabled 
			AND station.xCanRun 
			AND NOT fbMachine[1].xStopped 
			AND NOT station.xSingleRunning 
		THEN
			station.xDone:=TRUE;
		END_IF
		
		IF  station.xSingleRunning 
			OR station.xCanRun 
			AND NOT station.xDone 
			AND NOT station.xDisabled 
			AND NOT fbMachine[1].xStopped
		THEN
			station.xCycleEnable:=TRUE;
			station.xDone:= FALSE;  
			station.iStepAuto:= 10;
		END_IF
    10: //复位数据 
			arTonDelay[02](IN:= FALSE); 
		//	IF  station.xSingleRunning THEN
				 FOR i:=1 TO gc_ModuleProNo BY 1 DO
						 MEMSET(ADR(tsModuleProcess[i]),0,SIZEOF(tsModuleProcess[i]));
				 END_FOR
	//		END_IF
			station.iStepAuto:=20;
			
	20:////Restore_after_Estop_Process1 上载数据流程
			IF  station.xSingleRunning THEN //OR fbMachine[1].xTryRun THEN
					station.iStepAuto:= 50;
			ELSIF tsModuleProcess[1].xProcessNotStarted AND NOT  tsModuleProcess[1].xProcessStarted THEN
					station.iStepAuto :=21; (*process not started*)
			ELSIF  tsModuleProcess[1].xProcessStarted AND NOT  tsModuleProcess[1].xProcessCompleted THEN
				 station.iStepAuto := 21;(*process started*)
			ELSIF  tsModuleProcess[1].xProcessCompleted AND NOT tsModuleProcess[1].xQDataCompleted  THEN
					station.iStepAuto := 40 ;(*process completed*)
			ELSIF tsModuleProcess[1].xQDataCompleted THEN
					station.iStepAuto :=40;(*Qdata completed *)
			ELSE
					station.iStepAuto :=21; 
			END_IF	
	21://
				tsModuleProcess[1].xProcessNotStarted:=TRUE;
				station.iStepAuto:= 30;
				
	30://数据load 
		tsModuleProcess[1].xProcessStarted	:=TRUE;
		MEMCPY(ADR(arProcessDataStation[1]),ADR(arMainlineFixtureData[arCurFixtureNumStation[12]]),SIZEOF(arMainlineFixtureData[arCurFixtureNumStation[12]]));
		MEMCPY(ADR(arProcessDataStation[2]),ADR(arMainlineFixtureData[arCurFixtureNumStation[13]]),SIZEOF(arMainlineFixtureData[arCurFixtureNumStation[13]]));
		tsModuleProcess[1].xProcessCompleted:=TRUE;
		tsModuleProcess[1].xQDataCompleted:=TRUE;
		station.iStepAuto:= 40;
	40: //判断产品状态
			IF	NOT fbMachine[1].xTryRun THEN
								 IF  station.xEmptyDone THEN
													 station.iStepAuto:= 999;	
								 ELSIF  arProcessDataStation[1].stProduct.xEmptying  AND 
												arProcessDataStation[2].stProduct.xEmptying  THEN
													 station.xEmptying:=TRUE;
													 station.iStepAuto:= 1000;
								 ELSIF  arProcessDataStation[1].xMaterialOnOff   AND
												arProcessDataStation[2].xMaterialOnOff  THEN
													 station.iStepAuto:= 50;
								 ELSIF	 NOT arProcessDataStation[1].xMaterialOnOff   AND
												NOT arProcessDataStation[2].xMaterialOnOff  THEN
													 station.iStepAuto:= 999;
								 END_IF
			 ELSE
			 			station.iStepAuto:= 50;
			 END_IF
	/////产品流程开始	
	50:////Restore_after_Estop_Process2 调整流程
			IF  station.xSingleRunning OR fbMachine[1].xTryRun THEN
					station.iStepAuto :=60; 
			ELSIF tsModuleProcess[2].xProcessNotStarted AND NOT  tsModuleProcess[2].xProcessStarted THEN
					station.iStepAuto :=60; (*process not started*)
			ELSIF  tsModuleProcess[2].xProcessStarted AND NOT  tsModuleProcess[2].xProcessCompleted THEN
				 station.iStepAuto := 60;(*process started*)
			ELSIF  tsModuleProcess[2].xProcessCompleted AND NOT tsModuleProcess[2].xQDataCompleted  THEN
					station.iStepAuto :=110;(*process completed*)
			ELSIF tsModuleProcess[2].xQDataCompleted THEN
					station.iStepAuto :=200;(*Qdata completed *)
			ELSE
					station.iStepAuto :=60; 
			END_IF	
	60://等待
				 tsModuleProcess[2].xProcessNotStarted:=TRUE;
							 station.iStepAuto :=70; 
	70://Z轴伺服下降
			 tsModuleProcess[2].xProcessStarted:=TRUE;
			fbZAxisMove_1.xMoveAuto[2]:=TRUE;
		    fbZAxisMove_2.xMoveAuto[2]:=TRUE;
			IF  fbZAxisMove_1.xMoveInPos[2] AND fbZAxisMove_2.xMoveInPos[2] THEN
				station.iStepAuto:=80;	
			END_IF
	80://复位延时
				arTonDelay[02](IN:= FALSE); 
					station.iStepAuto:=90;
	90://延时等待
		arTonDelay[02](IN:= TRUE , PT:=T#2S , Q=> , ET=>);//伺服下压延时		
		IF  arTonDelay[2].Q THEN
			station.iStepAuto:=100;
		END_IF
		
	100://Z轴伺服上升
			fbZAxisMove_1.xMoveAuto[1]:=TRUE;
		    fbZAxisMove_2.xMoveAuto[1]:=TRUE;
		IF  fbZAxisMove_1.xMoveInPos[1] AND fbZAxisMove_2.xMoveInPos[1] THEN
			station.iStepAuto:=110;	
		END_IF	
	110:
		 tsModuleProcess[2].xProcessCompleted:=TRUE;
		 station.iStepAuto:=120;	
	120://调整结果
		arProcessDataStation[1].stProduct.xAdjusting_NOK:=FALSE;
		arProcessDataStation[2].stProduct.xAdjusting_OK :=TRUE;
		 tsModuleProcess[2].xQDataCompleted:=TRUE;
		station.iStepAuto:=200;
	
	////产品流程结束	
	200:////Restore_after_Estop_Process3 数据传输流程
			IF  station.xSingleRunning  THEN //OR fbMachine[1].xTryRun THEN
					station.iStepAuto :=999;
			ELSIF tsModuleProcess[3].xProcessNotStarted AND NOT  tsModuleProcess[3].xProcessStarted THEN
					station.iStepAuto :=210; (*process not started*)
			ELSIF  tsModuleProcess[3].xProcessStarted AND NOT  tsModuleProcess[3].xProcessCompleted THEN
				 station.iStepAuto := 220;(*process started*)
			ELSIF  tsModuleProcess[3].xProcessCompleted AND NOT tsModuleProcess[3].xQDataCompleted  THEN
					station.iStepAuto :=230;(*process completed*)
			ELSIF tsModuleProcess[3].xQDataCompleted THEN
					station.iStepAuto :=999;(*Qdata completed *)
			ELSE
					station.iStepAuto :=210; 
			END_IF		
	210://		
			tsModuleProcess[3].xProcessNotStarted:=TRUE;
			station.iStepAuto :=220; 
	220://数据unload
			tsModuleProcess[3].xProcessStarted:=TRUE;
			MEMCPY(ADR(arMainlineFixtureData[arCurFixtureNumStation[12]]),ADR(arProcessDataStation[1]),SIZEOF(arProcessDataStation[1]));
			MEMCPY(ADR(arMainlineFixtureData[arCurFixtureNumStation[13]]),ADR(arProcessDataStation[2]),SIZEOF(arProcessDataStation[2]));
			station.iStepAuto:= 230;
	230://
			tsModuleProcess[3].xProcessCompleted:=TRUE;
			station.iStepAuto :=240; 
 	240://本地数据清除
	//		MEMSET(ADR(arProcessDataStation[1]),0,SIZEOF(arProcessDataStation[1]));
	//		MEMSET(ADR(arProcessDataStation[2]),0,SIZEOF(arProcessDataStation[2]));
			tsModuleProcess[3].xQDataCompleted:=TRUE;
			station.iStepAuto:= 999;
	999://----Single Run Finish----
			
		station.iStepAuto :=0;
		IF NOT station.xSingleContinuousRun THEN
			station.xSingleRunFlag:=FALSE;
		END_IF
		station.xCycleEnable:=FALSE;	
		station.xDone:=TRUE;

{region "清料程序"}
1000://写入数据
	 		arProcessDataStation[1].xMaterialOnOff:=FALSE;
			arProcessDataStation[2].xMaterialOnOff:=FALSE;
	 		arProcessDataStation[1].stProduct.xAdjusting_NOK:=FALSE;
			arProcessDataStation[2].stProduct.xAdjusting_OK:=FALSE;
			arProcessDataStation[1].stProduct.xAdjusting_NOK:=FALSE;
			arProcessDataStation[2].stProduct.xAdjusting_OK:=FALSE;
			arProcessDataStation[1].stProduct.xEmptying:=TRUE;
			arProcessDataStation[2].stProduct.xEmptying:=TRUE;
			MEMCPY(ADR(arMainlineFixtureData[arCurFixtureNumStation[12]]),ADR(arProcessDataStation[1]),SIZEOF(arProcessDataStation[1]));
			MEMCPY(ADR(arMainlineFixtureData[arCurFixtureNumStation[13]]),ADR(arProcessDataStation[2]),SIZEOF(arProcessDataStation[2]));
			station.iStepAuto:= 1010;
1010://Z轴回参考位置
			fbZAxisMove_1.xMoveAuto[1]:=TRUE;
			fbZAxisMove_2.xMoveAuto[1]:=TRUE;
			IF  fbZAxisMove_1.xMoveInPos[1] AND fbZAxisMove_2.xMoveInPos[1]THEN
				station.iStepAuto:=1020;	
			END_IF	 
1020://清料完成
	 		station.xEmptying:=FALSE;
		  station.xEmptyDone:=TRUE;
			station.iStepAuto:=0;
{endRegion}	
		
				
		
		
		
		
		
		
		
		
		
	ELSE
		;	
END_CASE

END_IF
END_ACTION

ACTION FlowInit:
IF NOT station.xIniting THEN
  station.iStepInit:=0;    
ELSE
//--------------------------------------------初始化步序----------------------------------
CASE station.iStepInit OF	
 0://  
  	IF station.xIniting THEN	
  	  station.iStepInit:=10;	
  	END_IF	
10://复位数据
	FOR i:=1 TO gc_ModuleProNo BY 1 DO
				MEMSET(ADR(tsModuleProcess[i]),0,SIZEOF(tsModuleProcess[i]));
		END_FOR
	station.iStepInit:=20;
20://伺服上电
	fbZAxisMove_1.xPowerInit:=TRUE;
    fbZAxisMove_2.xPowerInit:=TRUE;
	IF  fbZAxisMove_1.xPowerOn AND fbZAxisMove_2.xPowerOn THEN
		station.iStepInit:=30;	
	END_IF
30://伺服去参考位位置
	fbZAxisMove_1.xMoveAuto[1]:=TRUE;
    fbZAxisMove_2.xMoveAuto[1]:=TRUE;
	IF  fbZAxisMove_1.xMoveInPos[1] AND fbZAxisMove_2.xMoveInPos[1] THEN
		station.iStepInit:=100;	
	END_IF
100://	
    station.iStepInit:=999;	
999://初始化完成	
	station.iStepInit:=0;
	station.xInitDone:=TRUE;  
END_CASE
END_IF
END_ACTION

ACTION General:
(******************清除过程记录**********************)
CASE bClearProcessStep OF
	0:	
		IF	 S08_MainLine.xClearProcessStatus THEN
			FOR i:=1 TO gc_ModuleProNo BY 1 DO
				MEMSET(ADR(tsModuleProcess[i]),0,SIZEOF(tsModuleProcess[i]));
			END_FOR
			bClearProcessStep:=10;
		END_IF
	10:
		xClearModuleProcessDone:=TRUE;
		bClearProcessStep:=20;
	20:
		IF NOT S08_MainLine.xClearProcessStatus THEN
			xClearModuleProcessDone:=FALSE;
			bClearProcessStep:=30;
		END_IF
	30:  
			bClearProcessStep:=0;
END_CASE
END_ACTION

ACTION ILC:

//---------------------------------------------------工站可执行-------------------------------------------------------
station.xCanRun :=TRUE ;

//---------------------------------------------------气缸动作条件-------------------------------------------


//---------------------------------------------------伺服动作条件-------------------------------------------

fbZAxisMove_1.xRunILC := 
fbZAxisMove_1.xMoveILC[1] :=
fbZAxisMove_1.xMoveILC[2] :=
fbZAxisMove_1.xMoveILC[3] :=
fbZAxisMove_1.xMoveILC[4] :=
fbZAxisMove_1.xMoveILC[5] := TRUE ;

fbZAxisMove_2.xRunILC := 
fbZAxisMove_2.xMoveILC[1] :=
fbZAxisMove_2.xMoveILC[2] :=
fbZAxisMove_2.xMoveILC[3] :=
fbZAxisMove_2.xMoveILC[4] :=
fbZAxisMove_2.xMoveILC[5] := TRUE ;
END_ACTION

ACTION TipAuto:

//------------------------------------------------AutoTip Cylinder--------------------------------

//------------------------------------------------AutoTip Servo--------------------------------
//**************************************
FOR i:= 1 TO 5 BY 1 DO 
	IF fbZAxisMove_1.xMoveAuto[i] THEN
		fbZAxisMove_1.iPosNumber := i ;
	END_IF
	IF fbZAxisMove_2.xMoveAuto[i] THEN
		fbZAxisMove_2.iPosNumber := i ;
	END_IF
	
END_FOR

IF  fbMachine[1].xAutoMode AND NOT fbMachine[1].xRunning  AND arTonDelay[09].Q  THEN 
	IF	fbZAxisMove_1.iPosNumber=1 	AND NOT fbZAxisMove_1.xMoveInPos[1] 	THEN 	station.adwAutoTip[1].10:=TRUE	;	END_IF//轴伺服自动时位置不在位置1
	if	fbZAxisMove_1.iPosNumber=2	AND NOT fbZAxisMove_1.xMoveInPos[2]	THEN 	station.adwAutoTip[1].11:=TRUE	;	END_IF//轴伺服自动时位置不在位置2
	if	fbZAxisMove_1.iPosNumber=3	AND NOT fbZAxisMove_1.xMoveInPos[3]	THEN 	station.adwAutoTip[1].12:=TRUE	;	END_IF//轴伺服自动时位置不在位置3
	if	fbZAxisMove_1.iPosNumber=4	AND NOT fbZAxisMove_1.xMoveInPos[4]	THEN 	station.adwAutoTip[1].13:=TRUE	;	END_IF//轴伺服自动时位置不在位置4
	IF	fbZAxisMove_1.iPosNumber=5	AND NOT fbZAxisMove_1.xMoveInPos[5]	THEN 	station.adwAutoTip[1].14:=TRUE	;	END_IF//轴伺服自动时位置不在位置5
END_IF
IF  fbMachine[1].xAutoMode AND NOT fbMachine[1].xRunning  AND arTonDelay[10].Q  THEN 
	IF	fbZAxisMove_2.iPosNumber=1 	AND NOT fbZAxisMove_2.xMoveInPos[1] 	THEN 	station.adwAutoTip[1].15:=TRUE	;	END_IF//轴伺服自动时位置不在位置1
	if	fbZAxisMove_2.iPosNumber=2	AND NOT fbZAxisMove_2.xMoveInPos[2]	THEN 	station.adwAutoTip[1].16:=TRUE	;	END_IF//轴伺服自动时位置不在位置2
	if	fbZAxisMove_2.iPosNumber=3	AND NOT fbZAxisMove_2.xMoveInPos[3]	THEN 	station.adwAutoTip[1].17:=TRUE	;	END_IF//轴伺服自动时位置不在位置3
	if	fbZAxisMove_2.iPosNumber=4	AND NOT fbZAxisMove_2.xMoveInPos[4]	THEN 	station.adwAutoTip[1].18:=TRUE	;	END_IF//轴伺服自动时位置不在位置4
	if	fbZAxisMove_2.iPosNumber=5	AND NOT fbZAxisMove_2.xMoveInPos[5]	THEN 	station.adwAutoTip[1].19:=TRUE	;	END_IF//轴伺服自动时位置不在位置5
END_IF
END_ACTION

ACTION TipManual:
//--------------------------------------------ManualTip------------------------------------------------------

//-------------------------------------------气缸提示---------------------------------------------------------




/////////////////////////////////////////////////////////////////////////////////////////////////////////////////
END_ACTION

ACTION Z_Output:
(**************************气缸输出********************************)
END_ACTION

END_PROGRAM

// ---- POUs/001_Station/S06_Cutting.TcPOU
PROGRAM S06_Cutting
VAR
	//工站
	station					: REFERENCE TO FB_Station:=fbstation[6];
	//气缸
	fbGlampCyl_1	:REFERENCE TO FB_Cylinder:=fbCylinder[24];	//	夹膜气缸（前）
	fbGlampCyl_2	:REFERENCE TO FB_Cylinder:=fbCylinder[25];	//	夹膜气缸（后）
	fbHOZReachedCyl_1	:REFERENCE TO FB_Cylinder:=fbCylinder[26];	//	水平到位气缸1
	fbHOZReachedCyl_2	:REFERENCE TO FB_Cylinder:=fbCylinder[27];	//	水平到位气缸2
	fbHOZCyl	:REFERENCE TO FB_Cylinder:=fbCylinder[28];	//	水平切膜气缸
	fbVTCAdjustCyl	:REFERENCE TO FB_Cylinder:=fbCylinder[29];	//	下方顶升调整气缸
	fbGlampAdjustCyl_1	:REFERENCE TO FB_Cylinder:=fbCylinder[30];	//	下方夹爪调整气缸1
	fbGlampAdjustCyl_2	:REFERENCE TO FB_Cylinder:=fbCylinder[31];	//	下方夹爪调整气缸2
	fbGlampAdjustCyl_3	:REFERENCE TO FB_Cylinder:=fbCylinder[32];	//	下方夹爪调整气缸3
	fbPressCyl_1				:REFERENCE TO FB_Cylinder:=fbCylinder[41];	//	压膜气缸1
	fbPressCyl_2				:REFERENCE TO FB_Cylinder:=fbCylinder[42];	//	压膜气缸2
	fbVTCCyl						:REFERENCE TO FB_Cylinder:=fbCylinder[43];	//	切膜垂直气缸
	
	//伺服
	fbROTAxisMove	 :REFERENCE TO FB_Axis:=fbAxis[14];	//	切膜工位丢膜伺服

	//延时
	arTonDelay :ARRAY[1..20] OF TON;
	//返回值
	UdiReturnValue :ARRAY[1..20] OF UDINT;
	//本地过程数据
	arProcessDataStation : ARRAY [1..3] OF DUT_MainlineFixture;
	i: INT;
	// 临时变量
	_FirstCycle:ARRAY[1..10] OF BOOL;
	// 循环计数
	bCounter: BYTE;
	// 结束循环
	bEndCounter: BYTE;
	//过程记录
	tsModuleProcess:ARRAY[1..gc_ModuleProNo] OF DUT_Process;
	xClearModuleProcessDone:BOOL;
	bClearProcessStep	:BYTE;

	// //废弃铝膜吹气电磁阀
	xScrapBlowValve: BOOL;
	// //废弃铝膜吹气步骤
	iScrapBlowStep: INT;
END_VAR

A_Input();
Alarm();
Delay();
FlowAuto();
FlowInit();
General();
ILC();
TipAuto();
TipManual();
Z_Output();

ACTION A_Input:
//气缸
fbGlampCyl_1.xWP_Sensor	:=	IxS06GlampCyl_1WP AND IxS06GlampCyl_3WP	;
fbGlampCyl_1.xHP_Sensor	:=	IxS06GlampCyl_1HP and IxS06GlampCyl_3HP	;
fbGlampCyl_2.xWP_Sensor	:=	IxS06GlampCyl_2WP and IxS06GlampCyl_4WP	;
fbGlampCyl_2.xHP_Sensor	:=	IxS06GlampCyl_2HP and IxS06GlampCyl_4HP	;
fbHOZReachedCyl_1.xWP_Sensor	:=	IxS06HOZReachedCyl_1WP	;
fbHOZReachedCyl_1.xHP_Sensor	:=	IxS06HOZReachedCyl_1HP	;
fbHOZReachedCyl_2.xWP_Sensor	:=	IxS06HOZReachedCyl_2WP	;
fbHOZReachedCyl_2.xHP_Sensor	:=	IxS06HOZReachedCyl_2HP	;
fbHOZCyl.xWP_Sensor	:=	IxS06HOZCyl_1WP	;
fbHOZCyl.xHP_Sensor	:=	IxS06HOZCyl_1HP	;
fbVTCAdjustCyl.xWP_Sensor	:=	IxS06VTCAdjustCylWP	;
fbVTCAdjustCyl.xHP_Sensor	:=	IxS06VTCAdjustCylHP	;
fbGlampAdjustCyl_1.xWP_Sensor	:= NOT 	IxS06GlampAdjustCyl_1HP AND arTonDelay[04].Q; //IxS06GlampAdjustCyl_1WP	;
fbGlampAdjustCyl_1.xHP_Sensor	:=	IxS06GlampAdjustCyl_1HP	;
fbGlampAdjustCyl_2.xWP_Sensor	:=	NOT IxS06GlampAdjustCyl_2HP AND arTonDelay[05].Q;//IxS06GlampAdjustCyl_2WP	;
fbGlampAdjustCyl_2.xHP_Sensor	:=	IxS06GlampAdjustCyl_2HP	;
fbGlampAdjustCyl_3.xWP_Sensor	:=	NOT IxS06GlampAdjustCyl_3HP AND arTonDelay[06].Q;//IxS06GlampAdjustCyl_3WP	;
fbGlampAdjustCyl_3.xHP_Sensor	:=	IxS06GlampAdjustCyl_3HP	;

fbPressCyl_1.xWP_Sensor:=IxS06PressCyl_1HP	;
fbPressCyl_1.xHP_Sensor:=IxS06PressCyl_1WP	;
fbPressCyl_2.xWP_Sensor:=IxS06PressCyl_2HP	;
fbPressCyl_2.xHP_Sensor:=IxS06PressCyl_2WP	;
fbVTCCyl.xWP_Sensor:=	   IxS06VTCCylHP	;
fbVTCCyl.xHP_Sensor:=	   IxS06VTCCylWP	;
END_ACTION

ACTION Alarm:
station.adwAlarm[1].00	:=	station.xInitTimeout	;//	S06 初始化超时
station.adwAlarm[1].01	:=	fbGlampCyl_2.xHP_Off	;//	S06切膜工位夹膜气缸(前)原点未到位
station.adwAlarm[1].02	:=	fbGlampCyl_1.xWP_Off	;//	S06切膜工位夹膜气缸(前)动点未到位
station.adwAlarm[1].03	:=	fbGlampCyl_2.xHP_Off	;//	S06切膜工位夹膜气缸(后)原点未到位
station.adwAlarm[1].04	:=	fbGlampCyl_2.xWP_Off	;//	S06切膜工位夹膜气缸(后)动点未到位
station.adwAlarm[1].05	:=	fbHOZReachedCyl_1.xHP_Off 	;//	S06切膜工位水平到位气缸1原点未到位
station.adwAlarm[1].06	:=	fbHOZReachedCyl_1.xWP_Off	;//	S06切膜工位水平到位气缸1动点未到位
station.adwAlarm[1].07	:=	fbHOZReachedCyl_2.xHP_Off	;//	S06切膜工位水平到位气缸2原点未到位
station.adwAlarm[1].08	:=	fbHOZReachedCyl_2.xWP_Off	;//	S06切膜工位水平到位气缸2动点未到位
station.adwAlarm[1].09	:=	fbHOZCyl.xHP_Off 	;//	S06切膜工位水平切膜气缸原点未到位
station.adwAlarm[1].10	:=	fbHOZCyl.xWP_Off 	;//	S06切膜工位水平切膜气缸动点未到位
station.adwAlarm[1].11	:=	fbVTCAdjustCyl.xHP_Off 	;//	S06切膜工位顶升气缸原点未到位
station.adwAlarm[1].12	:=	fbVTCAdjustCyl.xWP_Off 	;//	S06切膜工位顶升气缸动点未到位
station.adwAlarm[1].13	:=	fbGlampAdjustCyl_1.xHP_Off 	;//	S06切膜工位调整夹爪气缸1原点未到位
station.adwAlarm[1].14	:=	fbGlampAdjustCyl_1.xWP_Off	;//	S06切膜工位调整夹爪气缸1动点未到位
station.adwAlarm[1].15	:=	fbGlampAdjustCyl_2.xHP_Off	;//	S06切膜工位调整夹爪气缸2原点未到位
station.adwAlarm[1].16	:=	fbGlampAdjustCyl_2.xWP_Off	;//	S06切膜工位调整夹爪气缸2动点未到位
station.adwAlarm[1].17	:=	fbGlampAdjustCyl_3.xHP_Off	;//	S06切膜工位调整夹爪气缸3原点未到位
station.adwAlarm[1].18	:=	fbGlampAdjustCyl_3.xWP_Off	;//	S06切膜工位调整夹爪气缸3动点未到位
END_ACTION

ACTION Delay:
arTonDelay[01](IN:= , PT:=T#0.1S , Q=> , ET=> );
arTonDelay[02](IN:=  , PT:=T#1S , Q=> , ET=> );
arTonDelay[03](IN:=   , PT:=T#1S , Q=> , ET=> );
arTonDelay[04](IN:= fbGlampAdjustCyl_1.xWP_Valve AND  NOT IxS06GlampAdjustCyl_1HP, PT:=T#500MS , Q=> , ET=> );
arTonDelay[05](IN:= fbGlampAdjustCyl_2.xWP_Valve AND  NOT IxS06GlampAdjustCyl_2HP, PT:=T#500MS , Q=> , ET=> );
arTonDelay[06](IN:= fbGlampAdjustCyl_3.xWP_Valve AND  NOT IxS06GlampAdjustCyl_3HP, PT:=T#500MS , Q=> , ET=> );
arTonDelay[07](IN:= , PT:=T#0.1S , Q=> , ET=> );
arTonDelay[08](IN:= , PT:=T#0.1S , Q=> , ET=> );
arTonDelay[09](IN:= , PT:=T#0.1S , Q=> , ET=> );//铝膜吹气已使用
arTonDelay[10](IN:= NOT fbROTAxisMove.xbusy , PT:=T#0.1S , Q=> , ET=> );//TipAuto使用
END_ACTION

ACTION FlowAuto:

//-----------------------------------------初始化是否完成判断----------------------------------------------
IF NOT station.xInitDone 
THEN
 	station.iStepAuto:=0;
 	station.xDone:=FALSE;
ELSIF station.xRunning OR (  tsModuleProcess[2].xProcessStarted AND   NOT tsModuleProcess[2].xProcessCompleted)
THEN
//-----------------------------------------动作步骤--------------------------------------------------------
CASE station.iStepAuto OF	  
	0: //----Home Step，等待启动----
		IF station.xDisabled 
			AND station.xCanRun 
			AND NOT fbMachine[1].xStopped 
			AND NOT station.xSingleRunning 
		THEN
			station.xDone:=TRUE;
		END_IF
		
		IF  station.xSingleRunning 
			OR station.xCanRun 
			AND NOT station.xDone 
			AND NOT station.xDisabled 
			AND NOT fbMachine[1].xStopped
		THEN
			station.xCycleEnable:=TRUE;
			station.xDone:= FALSE;  
			station.iStepAuto:= 5;
		END_IF
    5: //复位数据 
			//	IF  station.xSingleRunning THEN
				 FOR i:=1 TO gc_ModuleProNo BY 1 DO
						 MEMSET(ADR(tsModuleProcess[i]),0,SIZEOF(tsModuleProcess[i]));
				 END_FOR
		//	END_IF
			station.iStepAuto:=10;
	10: //判断产品是否到该工位
		IF (* fbMachine[1].xTryRun OR*) station.xSingleRunning THEN
			station.iStepAuto:= 20;
		ELSE
		 	IF		station.xEmptyDone THEN
									station.iStepAuto:= 999;
			ELSIF	arMainlineFixtureData[arCurFixtureNumStation[14]].stProduct.xEmptying AND    
				    arMainlineFixtureData[arCurFixtureNumStation[15]].stProduct.xEmptying THEN
										station.xEmptying:=TRUE;
										station.iStepAuto:= 1000;
			ELSIF  NOT  arMainlineFixtureData[arCurFixtureNumStation[14]].xMaterialOnOff AND
						 NOT arMainlineFixtureData[arCurFixtureNumStation[15]].xMaterialOnOff AND 
						 NOT arMainlineFixtureData[arCurFixtureNumStation[16]].xMaterialOnOff THEN
										station.iStepAuto:= 999;			
			ELSIF	arMainlineFixtureData[arCurFixtureNumStation[14]].xMaterialOnOff AND    
				    arMainlineFixtureData[arCurFixtureNumStation[15]].xMaterialOnOff  THEN 
										station.iStepAuto:= 20;
			END_IF
		END_IF
	20:////Restore_after_Estop_Process1 上载数据流程
			IF  station.xSingleRunning  THEN //OR  fbMachine[1].xTryRun THEN
					station.iStepAuto :=40; 
			ELSIF tsModuleProcess[1].xProcessNotStarted AND NOT  tsModuleProcess[1].xProcessStarted THEN
					station.iStepAuto :=21; (*process not started*)
			ELSIF  tsModuleProcess[1].xProcessStarted AND NOT  tsModuleProcess[1].xProcessCompleted THEN
				 station.iStepAuto := 21;(*process started*)
			ELSIF  tsModuleProcess[1].xProcessCompleted AND NOT tsModuleProcess[1].xQDataCompleted  THEN
					station.iStepAuto := 40 ;(*process completed*)
			ELSIF tsModuleProcess[1].xQDataCompleted THEN
					station.iStepAuto :=40;(*Qdata completed *)
			ELSE
					station.iStepAuto :=21; 
			END_IF	
	21://
				tsModuleProcess[1].xProcessNotStarted:=TRUE;
				station.iStepAuto:= 30;
	30://上载产品数据
			tsModuleProcess[1].xProcessStarted	:=TRUE;
			IF  arMainlineFixtureData[arCurFixtureNumStation[14]].xMaterialOnOff  THEN
				MEMCPY(ADR(arProcessDataStation[1]),ADR(arMainlineFixtureData[arCurFixtureNumStation[14]]),SIZEOF(arMainlineFixtureData[arCurFixtureNumStation[14]]));
			END_IF
				MEMCPY(ADR(arProcessDataStation[2]),ADR(arMainlineFixtureData[arCurFixtureNumStation[15]]),SIZEOF(arMainlineFixtureData[arCurFixtureNumStation[15]]));
			IF  arMainlineFixtureData[arCurFixtureNumStation[16]].xMaterialOnOff THEN
				MEMCPY(ADR(arProcessDataStation[3]),ADR(arMainlineFixtureData[arCurFixtureNumStation[16]]),SIZEOF(arMainlineFixtureData[arCurFixtureNumStation[16]]));
			END_IF
			tsModuleProcess[1].xProcessCompleted:=TRUE;
			station.iStepAuto:= 40;			
	/////产品流程开始	
	40:
		station.iStepAuto:= 45;
	45://上方下压气缸伸出
			IF  arProcessDataStation[1].xMaterialOnOff THEN
						fbPressCyl_1.xAuto:=TRUE;
			END_IF
			IF   arProcessDataStation[3].xMaterialOnOff THEN
						fbPressCyl_2.xAuto:=TRUE;
			END_IF
		IF    ( fbPressCyl_1.xWP_Delay OR NOT  arProcessDataStation[1].xMaterialOnOff) AND
			  (fbPressCyl_2.xWP_Delay OR  NOT  arProcessDataStation[3].xMaterialOnOff)  THEN
				station.iStepAuto :=50;	
		END_IF		
	50://下方顶升气缸伸出
		fbVTCAdjustCyl.xAuto:=TRUE;
		IF fbVTCAdjustCyl.xWP_Delay THEN
			station.iStepAuto :=60;	
		END_IF	
	60://下方夹爪气缸夹紧
			IF  arProcessDataStation[1].xMaterialOnOff THEN
				fbGlampAdjustCyl_1.xAuto:=TRUE;
			END_IF
				fbGlampAdjustCyl_2.xAuto:=TRUE;
			IF   arProcessDataStation[3].xMaterialOnOff THEN
				fbGlampAdjustCyl_3.xAuto:=TRUE;
			END_IF
			IF    ( fbGlampAdjustCyl_1.xWP_Delay OR arProcessDataStation[1].xMaterialOnOff=FALSE) AND
				  fbGlampAdjustCyl_2.xWP_Delay  AND 
				  (fbGlampAdjustCyl_3.xWP_Delay OR  arProcessDataStation[3].xMaterialOnOff =FALSE)  THEN
					station.iStepAuto :=61;	
			END_IF
	61://上方下压气缸伸出
				IF  arProcessDataStation[1].xMaterialOnOff THEN
							fbPressCyl_1.xAuto:=TRUE;
				END_IF
				IF   arProcessDataStation[3].xMaterialOnOff THEN
							fbPressCyl_2.xAuto:=TRUE;
				END_IF
			IF    ( fbPressCyl_1.xWP_Delay OR NOT  arProcessDataStation[1].xMaterialOnOff) AND
				  (fbPressCyl_2.xWP_Delay OR  NOT  arProcessDataStation[3].xMaterialOnOff)  THEN
					station.iStepAuto :=65;	
			END_IF	
	65://允许调整工位动作
			//xS05WorkPermit:=TRUE;
			station.iStepAuto :=70;	
	70://水平到位气缸伸出
		fbHOZReachedCyl_1.xauto :=TRUE;
		fbHOZReachedCyl_2.xauto :=true;
		IF	fbHOZReachedCyl_1.xWP_Delay AND 
			fbHOZReachedCyl_2.xWP_Delay THEN
				station.iStepAuto :=80;	
		END_IF
	80://前后侧夹爪气缸夹住铝膜
		fbGlampCyl_1.xauto :=TRUE;
		fbGlampCyl_2.xauto:=TRUE;
		IF	fbGlampCyl_1.xWP_Delay AND 
			fbGlampCyl_2.xWP_Delay THEN
				station.iStepAuto :=90;	
		END_IF
	90:////Restore_after_Estop_Process2 切膜流程
			IF  station.xSingleRunning OR fbMachine[1].xTryRun THEN
					station.iStepAuto :=100; 
			ELSIF tsModuleProcess[2].xProcessNotStarted AND NOT  tsModuleProcess[2].xProcessStarted THEN
					station.iStepAuto :=110; (*process not started*)
			ELSIF  tsModuleProcess[2].xProcessStarted AND NOT  tsModuleProcess[2].xProcessCompleted THEN
				 station.iStepAuto := 110;(*process started*)
			ELSIF  tsModuleProcess[2].xProcessCompleted AND NOT tsModuleProcess[2].xQDataCompleted  THEN
					station.iStepAuto :=120;(*process completed*)
			ELSIF tsModuleProcess[2].xQDataCompleted THEN
					station.iStepAuto :=130;(*Qdata completed *)
			ELSE
					station.iStepAuto :=100; 
			END_IF	
	100://	
			 tsModuleProcess[2].xProcessNotStarted:=TRUE;
			 station.iStepAuto :=110; 
	
	110://切膜流程开始,垂直切膜气缸动作
			tsModuleProcess[2].xProcessStarted:=TRUE;
			fbVTCCyl.xAuto:=TRUE;
			IF fbVTCCyl.xWP_Delay THEN
			 		station.iStepAuto :=112;		
			END_IF
	112://正式切膜
			fbHOZCyl.xAuto:=TRUE;
			IF  fbHOZCyl.xWP_Delay THEN
				station.iStepAuto :=115;		
			END_IF
	115://水平切膜气缸返回
				fbHOZCyl.xAuto:=FALSE;
			IF  fbHOZCyl.xHP_Delay THEN
				station.iStepAuto :=116;		
			END_IF	
	116://切膜垂直气缸收回
				fbVTCCyl.xAuto:=FALSE;
			IF fbVTCCyl.xHP_Delay THEN
			 		station.iStepAuto :=120;		
			END_IF
	120:
			tsModuleProcess[2].xProcessCompleted:=TRUE;
			station.iStepAuto :=125;	
	125:	
		IF  arProcessDataStation[1].xMaterialOnOff  THEN
			arProcessDataStation[1].stProduct.xCutting_NOK:=FALSE;
			arProcessDataStation[1].stProduct.xCutting_OK:=TRUE;		
		END_IF
		
		arProcessDataStation[2].stProduct.xCutting_NOK:=FALSE;
		arProcessDataStation[2].stProduct.xCutting_OK:=TRUE;
		
		IF  arProcessDataStation[3].xMaterialOnOff  THEN
			arProcessDataStation[3].stProduct.xCutting_NOK:=FALSE;
			arProcessDataStation[3].stProduct.xCutting_OK:=TRUE;		
		END_IF
		tsModuleProcess[2].xQDataCompleted:=TRUE;
		station.iStepAuto :=130;	
	
	130://后侧夹爪气缸松开
			fbGlampCyl_2.xauto:=FALSE;
			IF	fbGlampCyl_2.xHP_Delay THEN
					station.iStepAuto :=140;	
			END_IF
	140://水平到位气缸收回
			fbHOZReachedCyl_1.xauto :=FALSE;
			fbHOZReachedCyl_2.xauto :=FALSE;
			IF	fbHOZReachedCyl_1.xHP_Delay AND 
				fbHOZReachedCyl_2.xHP_Delay THEN
					station.iStepAuto :=150;	
			END_IF	
	150://旋转伺服去工作位置
		 fbROTAxisMove.xMoveAuto[2]:=TRUE;
		
		 IF fbROTAxisMove.xMoveInPos[2] THEN
			 xScrapBlowValve:=TRUE;//废弃铝膜吹气打开
			 station.iStepAuto :=170; 
		 END_IF
//	155://垂直切膜气缸上升
//				fbVTCCyl.xAuto:=FALSE;
//			IF  fbVTCCyl.xHP_Delay THEN
//				station.iStepAuto :=170;		
//			END_IF 
//	//160://水平切膜气缸返回
	//	 	fbHOZCyl.xAuto:=FALSE;
	//		IF  fbHOZCyl.xHP_Delay THEN
	//			station.iStepAuto :=170;		
	//		END_IF 
	170://调整夹爪气缸松开
				
				fbGlampAdjustCyl_1.xAuto:=FALSE;
				fbGlampAdjustCyl_2.xAuto:=FALSE;
				fbGlampAdjustCyl_3.xAuto:=FALSE;
			IF   fbGlampAdjustCyl_1.xHP_Delay AND
				  fbGlampAdjustCyl_2.xHP_Delay  AND 
				  fbGlampAdjustCyl_3.xHP_Delay   THEN
					station.iStepAuto :=180;	
			END_IF
	180://顶升调整气缸收回
				fbVTCAdjustCyl.xAuto:=FALSE;
		IF fbVTCAdjustCyl.xHP_Delay THEN
			station.iStepAuto :=190;	
		END_IF	
	190://压膜气缸回原
			fbPressCyl_1.xAuto:=FALSE;
			fbPressCyl_2.xAuto:=FALSE;
			IF fbPressCyl_1.xHP_Delay AND 	
				 fbPressCyl_2.xHP_Delay  THEN
				station.iStepAuto :=200;	
			END_IF	
	////产品流程结束	
	200:////Restore_after_Estop_Process3 数据传输流程
			IF  station.xSingleRunning THEN // OR fbMachine[1].xTryRun THEN
					station.iStepAuto :=250;
			ELSIF tsModuleProcess[3].xProcessNotStarted AND NOT  tsModuleProcess[3].xProcessStarted THEN
					station.iStepAuto :=210; (*process not started*)
			ELSIF  tsModuleProcess[3].xProcessStarted AND NOT  tsModuleProcess[3].xProcessCompleted THEN
				 station.iStepAuto := 220;(*process started*)
			ELSIF  tsModuleProcess[3].xProcessCompleted AND NOT tsModuleProcess[3].xQDataCompleted  THEN
					station.iStepAuto :=230;(*process completed*)
			ELSIF tsModuleProcess[3].xQDataCompleted THEN
					station.iStepAuto :=250;(*Qdata completed *)
			ELSE
					station.iStepAuto :=210; 
			END_IF		
	210://		
				tsModuleProcess[3].xProcessNotStarted:=TRUE;
				station.iStepAuto :=220; 
	220://数据unload
		tsModuleProcess[3].xProcessStarted:=TRUE;
		IF arProcessDataStation[1].xMaterialOnOff  THEN
			MEMCPY(ADR(arMainlineFixtureData[arCurFixtureNumStation[14]]),ADR(arProcessDataStation[1]),SIZEOF(arProcessDataStation[1]));
		END_IF
		  MEMCPY(ADR(arMainlineFixtureData[arCurFixtureNumStation[15]]),ADR(arProcessDataStation[2]),SIZEOF(arProcessDataStation[2]));
		IF arProcessDataStation[3].xMaterialOnOff  THEN
			MEMCPY(ADR(arMainlineFixtureData[arCurFixtureNumStation[16]]),ADR(arProcessDataStation[3]),SIZEOF(arProcessDataStation[3]));
		END_IF
		station.iStepAuto:= 230;
	230://
			tsModuleProcess[3].xProcessCompleted:=TRUE;
			station.iStepAuto :=240; 
 	240://本地数据清除
	//		MEMSET(ADR(arProcessDataStation[1]),0,SIZEOF(arProcessDataStation[1]));
	//		MEMSET(ADR(arProcessDataStation[2]),0,SIZEOF(arProcessDataStation[2]));
	//		MEMSET(ADR(arProcessDataStation[3]),0,SIZEOF(arProcessDataStation[3]));
	//		tsModuleProcess[3].xQDataCompleted:=TRUE;
			station.iStepAuto:= 250;
	250://
				station.xDone:=TRUE;
				station.iStepAuto:= 260;
				
	260://夹爪松开			
			fbGlampCyl_1.xauto:=FALSE;
			IF	fbGlampCyl_1.xHP_Delay THEN
					station.iStepAuto :=270;	
			END_IF
	270://伺服回初始位置		
			fbROTAxisMove.xMoveAuto[1]:=TRUE;
		 IF fbROTAxisMove.xMoveInPos[1] THEN
			 station.iStepAuto :=999; 
		 END_IF
	999://----Single Run Finish----
			
		station.iStepAuto :=0;
		IF NOT station.xSingleContinuousRun THEN
			station.xSingleRunFlag:=FALSE;
		END_IF
		
		station.xCycleEnable:=FALSE;	
		station.xDone:=TRUE;	
		
		
{region "清料程序"}
1000://写入数据
	 		arProcessDataStation[1].xMaterialOnOff:=FALSE;
			arProcessDataStation[2].xMaterialOnOff:=FALSE;
			arProcessDataStation[3].xMaterialOnOff:=FALSE;
	 		arProcessDataStation[1].stProduct.xCutting_NOK:=FALSE;
			arProcessDataStation[1].stProduct.xCutting_OK:=FALSE;	
			arProcessDataStation[2].stProduct.xCutting_NOK:=FALSE;
			arProcessDataStation[2].stProduct.xCutting_OK:=FALSE;	
			arProcessDataStation[3].stProduct.xCutting_NOK:=FALSE;
			arProcessDataStation[3].stProduct.xCutting_OK:=FALSE;	
			arProcessDataStation[1].stProduct.xEmptying:=TRUE;
			arProcessDataStation[2].stProduct.xEmptying:=TRUE;
			arProcessDataStation[3].stProduct.xEmptying:=TRUE;
			MEMCPY(ADR(arMainlineFixtureData[arCurFixtureNumStation[14]]),ADR(arProcessDataStation[1]),SIZEOF(arProcessDataStation[1]));
			MEMCPY(ADR(arMainlineFixtureData[arCurFixtureNumStation[15]]),ADR(arProcessDataStation[2]),SIZEOF(arProcessDataStation[2]));
			MEMCPY(ADR(arMainlineFixtureData[arCurFixtureNumStation[16]]),ADR(arProcessDataStation[3]),SIZEOF(arProcessDataStation[3]));
			station.iStepAuto:= 1010;
1010://切莫垂直气缸收回
		fbVTCCyl.xAuto:=FALSE;
		IF  fbVTCCyl.xHP_Delay THEN
		 	station.iStepAuto :=1020;
		END_IF
1020://水平切膜气缸收回
		fbHOZCyl.xAuto:=FALSE;
		IF  fbHOZCyl.xHP_Delay THEN
			station.iStepAuto :=1030;
		END_IF
1030://后侧夹爪气缸松开
		fbGlampCyl_2.xauto :=FALSE;
		IF   fbGlampCyl_2.xHP_Delay THEN
			station.iStepAuto :=1040;
		END_IF
1040://水平对顶气缸收回
		fbHOZReachedCyl_1.xAuto :=FALSE;
		fbHOZReachedCyl_2.xAuto :=FALSE;
		IF   fbHOZReachedCyl_1.xHP_Delay AND
			 fbHOZReachedCyl_2.xHP_Delay THEN
			station.iStepAuto :=1050;
		END_IF	
1050://下压气缸回原
		fbPressCyl_1.xAuto :=FALSE;
		fbPressCyl_2.xAuto :=FALSE;
		IF  fbPressCyl_1.xHP_Delay  AND  
				fbPressCyl_2.xHP_Delay THEN
		 	station.iStepAuto :=1060;
		END_IF	
1060://旋转伺服旋转到位置1
		fbROTAxisMove.xMoveAuto[2]:=TRUE;
		IF  fbROTAxisMove.xMoveInPos[2] THEN
			station.iStepAuto :=1070;
		END_IF
1070://水平切莫气缸收回
		 fbHOZCyl.xAuto :=FALSE;
		 IF  fbHOZCyl.xHP_Delay THEN
				 station.iStepAuto :=1080;
		 END_IF
1080://前测夹爪气缸松开
		 fbGlampCyl_1.xAuto :=FALSE;
		 IF   fbGlampCyl_1.xHP_Delay THEN
			 station.iStepAuto :=1090;
		 END_IF
1090://旋转伺服回参考位置
		 fbROTAxisMove.xMoveAuto[1]:=TRUE;
		 IF  fbROTAxisMove.xMoveInPos[1] THEN
			 station.iStepAuto :=1100;
		 END_IF
1100://下方夹气缸松开
		 fbGlampAdjustCyl_1.xAuto :=FALSE;
		 fbGlampAdjustCyl_2.xAuto :=FALSE;
		 fbGlampAdjustCyl_3.xAuto :=FALSE;
	 IF fbGlampAdjustCyl_1.xHP_Delay AND 
		 fbGlampAdjustCyl_2.xHP_Delay AND 
			fbGlampAdjustCyl_3.xHP_Delay THEN
			station.iStepAuto :=1110;	
	 END_IF
1110://下方顶升气缸回原位
	fbVTCAdjustCyl.xAuto :=FALSE;
	IF fbVTCAdjustCyl.xHP_Delay THEN
		station.iStepAuto :=1120;	
	END_IF
1120://清料程序完成
			station.xEmptying:=FALSE;
			station.xEmptyDone:=TRUE;
			station.iStepAuto :=0;		 
{endregion}		
		
	ELSE
		;	
END_CASE



END_IF
END_ACTION

ACTION FlowInit:
IF NOT station.xIniting THEN
  station.iStepInit:=0;    
ELSE
//--------------------------------------------初始化步序----------------------------------
CASE station.iStepInit OF	
 0://  
  	IF station.xIniting THEN	
  	  station.iStepInit:=10;	
  	END_IF	
10://复位数据
	iScrapBlowStep:=0;
	FOR i:=1 TO gc_ModuleProNo BY 1 DO
				MEMSET(ADR(tsModuleProcess[i]),0,SIZEOF(tsModuleProcess[i]));
	END_FOR
	station.iStepInit :=20;
20://切莫垂直气缸收回
		fbVTCCyl.xInit:=TRUE;
		IF  fbVTCCyl.xHP_Delay THEN
		 	station.iStepInit :=40;
		END_IF
40://水平切膜气缸收回
	fbHOZCyl.xInit :=TRUE;
	IF  fbHOZCyl.xHP_Delay THEN
		station.iStepInit :=50;
	END_IF
50://后侧夹爪气缸松开
	fbGlampCyl_2.xInit :=TRUE;
	IF   fbGlampCyl_2.xHP_Delay THEN
		station.iStepInit :=60;
	END_IF
60://水平对顶气缸收回
	fbHOZReachedCyl_1.xInit :=TRUE;
	fbHOZReachedCyl_2.xInit :=TRUE;
	IF   fbHOZReachedCyl_1.xHP_Delay AND
		 fbHOZReachedCyl_2.xHP_Delay THEN
		station.iStepInit :=65;
	END_IF	
65://下压气缸回原
		fbPressCyl_1.xInit:=TRUE;
		fbPressCyl_2.xInit:=TRUE;
		IF  fbPressCyl_1.xHP_Delay  AND  
				fbPressCyl_2.xHP_Delay THEN
		 	station.iStepInit :=70;
		END_IF	
70:	//旋转伺服上电
	fbROTAxisMove.xPowerInit:=TRUE;
	IF  fbROTAxisMove.xPowerOn THEN
		station.iStepInit :=80;
	END_IF
80://旋转伺服旋转到位置1
	fbROTAxisMove.xMoveAuto[2]:=TRUE;
	IF  fbROTAxisMove.xMoveInPos[2] THEN
	 	xScrapBlowValve:=TRUE;//废弃铝膜吹气打开
		station.iStepInit :=90;
	END_IF
90://水平切莫气缸收回
	fbHOZCyl.xInit:=TRUE;
	IF  fbHOZCyl.xHP_Delay THEN
			station.iStepInit :=100;
	END_IF
	
100://前测夹爪气缸松开
	fbGlampCyl_1.xInit :=TRUE;
	IF   fbGlampCyl_1.xHP_Delay THEN
		station.iStepInit :=250;
	END_IF
(*************流程未开始*****************)
200://水平切膜收回
	fbHOZCyl.xInit:=TRUE;
	IF  fbHOZCyl.xHP_Delay THEN
			station.iStepInit :=210;
	END_IF
210://前后夹爪气缸松开
	fbGlampCyl_1.xInit :=TRUE;
	fbGlampCyl_2.xInit :=TRUE;
	IF   fbGlampCyl_1.xHP_Delay AND
		  fbGlampCyl_2.xHP_Delay THEN
		station.iStepInit :=220;
	END_IF	
220://水平对位气缸收回
	fbHOZReachedCyl_1.xInit :=TRUE;
	fbHOZReachedCyl_2.xInit :=TRUE;
	IF   fbHOZReachedCyl_1.xHP_Delay AND 
		 fbHOZReachedCyl_2.xHP_Delay THEN
		station.iStepInit :=250;
	END_IF	

250://旋转伺服回参考位置
	fbROTAxisMove.xMoveAuto[1]:=TRUE;
	IF  fbROTAxisMove.xMoveInPos[1] THEN
		station.iStepInit :=260;
	END_IF
260://下方夹气缸松开
	fbGlampAdjustCyl_1.xinit :=TRUE;
    fbGlampAdjustCyl_2.xinit :=true;
    fbGlampAdjustCyl_3.xinit :=TRUE;
	IF fbGlampAdjustCyl_1.xHP_Delay AND 
		fbGlampAdjustCyl_2.xHP_Delay AND 
	   fbGlampAdjustCyl_3.xHP_Delay THEN
	   station.iStepInit :=270;	
	END_IF
270://下方顶升气缸回原位
	fbVTCAdjustCyl.xInit:=TRUE;
	IF fbVTCAdjustCyl.xHP_Delay THEN
		station.iStepInit :=300;	
	END_IF
	
300://	
    station.iStepInit:=999;	
999://初始化完成	
	station.iStepInit:=0;
	station.xInitDone:=TRUE;  
END_CASE
END_IF
END_ACTION

ACTION General:
(******************清除过程记录**********************)
CASE bClearProcessStep OF
	0:	
		IF	 S08_MainLine.xClearProcessStatus THEN
			FOR i:=1 TO gc_ModuleProNo BY 1 DO
				MEMSET(ADR(tsModuleProcess[i]),0,SIZEOF(tsModuleProcess[i]));
			END_FOR
			bClearProcessStep:=10;
		END_IF
	10:
		xClearModuleProcessDone:=TRUE;
		bClearProcessStep:=20;
	20:
		IF NOT S08_MainLine.xClearProcessStatus THEN
			xClearModuleProcessDone:=FALSE;
			bClearProcessStep:=30;
		END_IF
	30:  
			bClearProcessStep:=0;
	
END_CASE
END_ACTION

ACTION ILC:

//---------------------------------------------------工站可执行-------------------------------------------------------
station.xCanRun :=TRUE ;

//---------------------------------------------------气缸动作条件-------------------------------------------
fbGlampCyl_1.xOffILC	:=	TRUE	;
fbGlampCyl_1.xOnILC	:=	TRUE	;
fbGlampCyl_2.xOffILC	:=	TRUE	;
fbGlampCyl_2.xOnILC	:=	TRUE	;
fbHOZReachedCyl_1.xOffILC	:=	TRUE	;
fbHOZReachedCyl_1.xOnILC	:=	TRUE	;
fbHOZReachedCyl_2.xOffILC	:=	TRUE	;
fbHOZReachedCyl_2.xOnILC	:=	TRUE	;
fbHOZCyl.xOffILC	:=	TRUE	;
fbHOZCyl.xOnILC	:=	TRUE	;
fbVTCAdjustCyl.xOffILC	:=	TRUE	;
fbVTCAdjustCyl.xOnILC	:=	TRUE	;
fbGlampAdjustCyl_1.xOffILC	:=	TRUE	;
fbGlampAdjustCyl_1.xOnILC	:=	TRUE	;
fbGlampAdjustCyl_2.xOffILC	:=	TRUE	;
fbGlampAdjustCyl_2.xOnILC	:=	TRUE	;
fbGlampAdjustCyl_3.xOffILC	:=	TRUE	;
fbGlampAdjustCyl_3.xOnILC	:=	TRUE	;
fbVTCCyl.xOffILC:=TRUE;
fbVTCCyl.xOnILC:=TRUE;
fbPressCyl_1.xOffILC:=TRUE;
fbPressCyl_1.xOnILC:=TRUE;
fbPressCyl_2.xOffILC:=TRUE;
fbPressCyl_2.xOnILC:=TRUE;


//---------------------------------------------------伺服动作条件-------------------------------------------
fbROTAxisMove.xRunILC := TRUE;
fbROTAxisMove.xMoveILC[1] :=fbHOZReachedCyl_1.xHP_Delay AND fbHOZReachedCyl_2.xHP_Delay ;
END_ACTION

ACTION TipAuto:

//------------------------------------------------AutoTip Cylinder--------------------------------
//station.adwAutoTip[1].00	:=	fbGlampCyl_1.xAutoTip	;
//station.adwAutoTip[1].01	:=	fbGlampCyl_2.xAutoTip	;
//station.adwAutoTip[1].02	:=	fbHOZReachedCyl_1.xAutoTip	;
//station.adwAutoTip[1].03	:=	fbHOZReachedCyl_2.xAutoTip	;
//station.adwAutoTip[1].04	:=	fbHOZCyl.xAutoTip	;
//station.adwAutoTip[1].05	:=	fbVTCAdjustCyl.xAutoTip	;
//station.adwAutoTip[1].06	:=	fbGlampAdjustCyl_1.xAutoTip	;
//station.adwAutoTip[1].07	:=	fbGlampAdjustCyl_2.xAutoTip	;
//station.adwAutoTip[1].08	:=	fbGlampAdjustCyl_3.xAutoTip	;

//------------------------------------------------AutoTip Servo--------------------------------
//**************************************
FOR i:= 1 TO 5 BY 1 DO 
	IF fbROTAxisMove.xMoveAuto[i] THEN
		fbROTAxisMove.iPosNumber := i ;
	END_IF
	
END_FOR


IF  fbMachine[1].xAutoMode AND NOT fbMachine[1].xRunning  AND arTonDelay[10].Q THEN
		IF	fbROTAxisMove.iPosNumber=1 	AND NOT fbROTAxisMove.xMoveInPos[1] 	THEN 	station.adwAutoTip[1].10:=TRUE	;	END_IF//轴伺服自动时位置不在位置1
		if	fbROTAxisMove.iPosNumber=2	AND NOT fbROTAxisMove.xMoveInPos[2]	THEN 	station.adwAutoTip[1].11:=TRUE	;	END_IF//轴伺服自动时位置不在位置2
		if	fbROTAxisMove.iPosNumber=3	AND NOT fbROTAxisMove.xMoveInPos[3]	THEN 	station.adwAutoTip[1].12:=TRUE	;	END_IF//轴伺服自动时位置不在位置3
		if	fbROTAxisMove.iPosNumber=4	AND NOT fbROTAxisMove.xMoveInPos[4]	THEN 	station.adwAutoTip[1].13:=TRUE	;	END_IF//轴伺服自动时位置不在位置4
		if	fbROTAxisMove.iPosNumber=5	AND NOT fbROTAxisMove.xMoveInPos[5]	THEN 	station.adwAutoTip[1].14:=TRUE	;	END_IF//轴伺服自动时位置不在位置5
END_IF
END_ACTION

ACTION TipManual:
//--------------------------------------------ManualTip------------------------------------------------------

//-------------------------------------------气缸提示---------------------------------------------------------




/////////////////////////////////////////////////////////////////////////////////////////////////////////////////
END_ACTION

ACTION Z_Output:
(**************************气缸输出********************************)
QxS06GlampCyl_1WP	:=	fbGlampCyl_1.xWP_Valve	;
QxS06GlampCyl_1HP	:=	fbGlampCyl_1.xHP_Valve	;
QxS06GlampCyl_2WP	:=	fbGlampCyl_2.xWP_Valve	;
QxS06GlampCyl_2HP	:=	fbGlampCyl_2.xHP_Valve	;
QxS06HOZReachedCyl_1WP	:=	fbHOZReachedCyl_1.xWP_Valve	;
QxS06HOZReachedCyl_1HP	:=	fbHOZReachedCyl_1.xHP_Valve	;
QxS06HOZReachedCyl_2WP	:=	fbHOZReachedCyl_2.xWP_Valve	;
QxS06HOZReachedCyl_2HP	:=	fbHOZReachedCyl_2.xHP_Valve	;
QxS06HOZCyl_1WP	:=	fbHOZCyl.xWP_Valve	;
QxS06HOZCyl_1HP	:=	fbHOZCyl.xHP_Valve	;
QxS06VTCAdjustCylWP	:=	fbVTCAdjustCyl.xWP_Valve	;
QxS06VTCAdjustCylHP	:=	fbVTCAdjustCyl.xHP_Valve	;
QxS06GlampAdjustCyl_1WP	:=	fbGlampAdjustCyl_1.xWP_Valve	;
QxS06GlampAdjustCyl_1HP	:=	fbGlampAdjustCyl_1.xHP_Valve	;
QxS06GlampAdjustCyl_2WP	:=	fbGlampAdjustCyl_2.xWP_Valve	;
QxS06GlampAdjustCyl_2HP	:=	fbGlampAdjustCyl_2.xHP_Valve	;
QxS06GlampAdjustCyl_3WP	:=	fbGlampAdjustCyl_3.xWP_Valve	;
QxS06GlampAdjustCyl_3HP	:=	fbGlampAdjustCyl_3.xHP_Valve	;
QxS06PressCyl_1WP					:=		fbPressCyl_1.xWP_Valve;
QxS06PressCyl_1HP	    		:=    fbPressCyl_1.xHP_Valve;
QxS06PressCyl_2WP	    		:=    fbPressCyl_2.xWP_Valve;
QxS06PressCyl_2HP	    		:=    fbPressCyl_2.xHP_Valve;
QxS06VTCCylWP				   		:=    fbVTCCyl.xWP_Valve;
QxS06VTCCylHP	    				:=    fbVTCCyl.xHP_Valve;
//铝膜吹气电磁阀手动
IF  fbMachine[1].xManualMode THEN
		 IF  xS06AluBlowValve THEN
				QxS06BlowValve:=TRUE;
		 ELSE
				QxS06BlowValve:=FALSE;
		 END_IF
END_IF

//铝膜吹气电磁阀自动
//每次使能吹气2s
CASE  iScrapBlowStep OF
 0://等待信号
 		IF xScrapBlowValve THEN
		 	 QxS06BlowValve:=FALSE;
			 xScrapBlowValve:=FALSE;
			iScrapBlowStep:=iScrapBlowStep +1; 
		END_IF
  1://开始吹气
  		QxS06BlowValve:=TRUE;
			arTonDelay[09](IN:= TRUE, PT:=T#2S , Q=> , ET=> );
			IF arTonDelay[09].Q THEN
			 		arTonDelay[09](IN:= FALSE);
			 		iScrapBlowStep:=iScrapBlowStep +1; 
			END_IF
	2://吹气关闭
			QxS06BlowValve:=FALSE;
			iScrapBlowStep:=0;
END_CASE
END_ACTION

END_PROGRAM

// ---- POUs/001_Station/S07_BoxCarrying.TcPOU
PROGRAM S07_BoxCarrying
VAR
	//工站
	station					: REFERENCE TO FB_Station:=fbstation[7];
	//气缸

	//伺服
	fbNGStepMotor	 :REFERENCE TO FB_Axis:=fbAxis[19];	//	NG流道旋转部进
	//大寰夹爪
	fbClamp			 	:REFERENCE TO FB_RGI_14_Modbus:=fbRGI_14_Modbus[1];
	//图灵机械手
	fbRobot   :REFERENCE TO FB_TURINContorl:=fbTURINContorl[1];
	//延时
	arTonDelay :ARRAY[1..20] OF TON;
	//返回值
	UdiReturnValue :ARRAY[1..20] OF UDINT;
	//本地过程数据
	arProcessDataStation : ARRAY [1..3] OF DUT_MainlineFixture;
	i: INT;
	// 临时变量
	_FirstCycle:ARRAY[1..10] OF BOOL;
	// 循环计数
	bCounter: BYTE;
	// 结束循环
	bEndCounter: BYTE;
	//过程记录
	tsModuleProcess:ARRAY[1..gc_ModuleProNo] OF DUT_Process;
	xClearModuleProcessDone:BOOL;
	bClearProcessStep	:BYTE;
	//机械手循环次数
	bRobCounter: BYTE;
	//放料到卡片上
	xPutBoxInCardPosDone :BOOL;
	//buffer位置是否有产品
	xBufferPosCheckSensor: BOOL;
	//NG流道传感器
	xNGPosCheckSensor :ARRAY[1..3] OF BOOL;
	//允许机械手放料到NG流道
	xNGPutBoxPermit:BOOL;
//	//入料线体深孔板检测
//	xBeltBoxCheckSensor:ARRAY[1..2] OF BOOL;
	//NG流道步骤
	iNGStep: INT;
	// //报警屏蔽
	_AlarmDisable: BOOL;
	//取上来的孔板放置位置
	iPutPartPosChoose:WORD;
	iPickPartPosChoose:WORD;
//	//已经放完的孔板位置
//	xPutBeltLineCompleted:ARRAY[1..2] OF BOOL;
	//主流线传感器
	xMainLineSensorReached:ARRAY[1..2] OF BOOL;

	// 临时
	bRobotStep: BYTE;
	// 临时
	xRobotStartTryRun: BOOL;
	test: BOOL;
	EstopR_TRIG: R_TRIG;
	MachineInitR_TRIG: R_TRIG;
	_FirstPosChoose: WORD;
	_SecondPosChoose: WORD;
	// 皮带线控制Done信号
	xBeltLineControl: BOOL;
	// NG流道允许运行
	xNGLinePremit: BOOL;
END_VAR

A_Input();
Alarm();
Delay();
FlowAuto();
FlowInit();
General();
ILC();
TipAuto();
TipManual();
Z_Output();

ACTION A_Input:
//传感器
xBufferPosCheckSensor:=IxBufferCheckSensor1;(*缓冲工位传感器*)
xNGPosCheckSensor[1]:=IxS07CheckSensor3;	(*NG流道传感器，机械手放料检测*)
xNGPosCheckSensor[2]:=IxS07CheckSensor2;	(*NG流道传感器,中间传感器**)
xNGPosCheckSensor[3]:=IxS07CheckSensor1; 	(*NG流道传感器，满料传感器*)


xMainLineSensorReached[1]:=IxLineEndSensor1Reached	;//	主流线尾端¶到位检测传感器1
xMainLineSensorReached[2]:=IxLineEndSensor2Reached	;//	主流线尾端¶到位检测传感器2

////入料线体深孔板检测
//xBeltBoxCheckSensor[1]:=IxBeltEntryBoxCheckSensor1	;
//xBeltBoxCheckSensor[2]:=IxBeltEntryBoxCheckSensor2	;
//
END_ACTION

ACTION Alarm:
//
station.adwAlarm[1].00:=station.xInitTimeout;	  			//S07BoxCarrying 初始化超时

(*station.adwAlarm[1].01:=TRUE;*)//NG流道满料请处理	  	
(*station.adwAlarm[1].02:=TRUE;*)//NG流道步进运动超时 ，请检查传感器是否正常
//station.adwAlarm[1].03	:=	fbRobot.eErrID<>0	;//	S07孔板搬运工位机械手报错
station.adwAlarm[1].04	:=	fbClamp.xError	;//	S07孔板搬运工位夹爪报错
//station.adwAlarm[1].05	:=	fbNGStepMotor.xError	;//	S07孔板搬运工位NG流道伺服报错
//station.adwAlarm[1].06	:=	fbNGStepMotor.xNotPowerOn	;//	S07孔板搬运工位NG流道伺服未使能
//station.adwAlarm[1].07	:=	fbNGStepMotor.xMoveTimeout	;//	S07孔板搬运工位NG流道伺服移动超时
IF 	station.xRunning AND	xMainLineSensorReached[2]  THEN 	
	arTonDelay[03](IN:= TRUE   , PT:=T#1S , Q=> , ET=> );
	IF  arTonDelay[03].Q THEN 
				station.adwAlarm[1].08	:=	TRUE 	;//	主流线结尾处检测到深孔板，请检查
	END_IF
ELSE
 arTonDelay[03](IN:= FALSE);
END_IF
//station.adwAlarm[1].09	:=	true	;//	S07孔板搬运工位卡片1位置不可重复放置,请检查
//station.adwAlarm[1].10	:=	true;//	S07孔板搬运工位卡片2位置不可重复放置,请检查
//station.adwAlarm[1].11	:=	true	;//	S07孔板搬运工位Buffer位置不可重复放置,请检查
//station.adwAlarm[1].12	:=	true	;//	S07孔板搬运工位NG位置不可重复放置,请检查


station.adwAlarm[1].13:= (station.xIniting AND NOT stFromRobot.xLocal_Remote)  ;//S07孔板搬运工位机械手示教器未打到自动模式
END_ACTION

ACTION Delay:
arTonDelay[01](IN:= , PT:=T#0.1S , Q=> , ET=> );
(*arTonDelay[02](IN:=  , PT:=T#1S , Q=> , ET=> );*)//NG流道使用
arTonDelay[03](IN:=   , PT:=T#1S , Q=> , ET=> );//尾端传感器报警用
arTonDelay[04](IN:= , PT:=T#0.1S , Q=> , ET=> );
arTonDelay[05](IN:= , PT:=T#0.1S , Q=> , ET=> );
arTonDelay[06](IN:= , PT:=T#0.1S , Q=> , ET=> );
arTonDelay[07](IN:= , PT:=T#0.1S , Q=> , ET=> );
arTonDelay[08](IN:= , PT:=T#0.1S , Q=> , ET=> );
arTonDelay[09](IN:= , PT:=T#0.1S , Q=> , ET=> );
arTonDelay[10](IN:= NOT fbNGStepMotor.xbusy  , PT:=T#0.1S , Q=> , ET=> );//TipAuto使用
END_ACTION

ACTION FlowAuto:
//-----------------------------------------初始化是否完成判断----------------------------------------------
IF NOT station.xInitDone 
THEN
 	station.iStepAuto:=0;
 	station.xDone:=FALSE;
ELSIF station.xRunning  OR ( tsModuleProcess[bRobCounter+1].xProcessStarted AND NOT   tsModuleProcess[bRobCounter+1].xProcessCompleted) OR
 												 ( tsModuleProcess[bRobCounter+3].xProcessStarted AND NOT   tsModuleProcess[bRobCounter+3].xProcessCompleted)
THEN
//-----------------------------------------动作步骤--------------------------------------------------------
CASE station.iStepAuto OF	  
	0: //----Home Step，等待启动----
		IF station.xDisabled 
			AND station.xCanRun 
			AND NOT fbMachine[1].xStopped 
			AND NOT station.xSingleRunning 
		THEN
			station.xDone:=TRUE;
			xS07MainlineRunPermit:=TRUE;
		END_IF
		
		IF  station.xSingleRunning 
			OR station.xCanRun 
			//AND NOT station.xDone 
			AND NOT station.xDisabled 
			AND NOT fbMachine[1].xStopped
		THEN
			station.xCycleEnable:=TRUE;
			//station.xDone:= FALSE;  
			station.iStepAuto:= 5;
		END_IF
    5: //复位数据
			IF  station.xSingleRunning THEN
				 FOR i:=1 TO gc_ModuleProNo BY 1 DO
						 MEMSET(ADR(tsModuleProcess[i]),0,SIZEOF(tsModuleProcess[i]));
				 END_FOR
			END_IF
			station.iStepAuto:=10;
	10: //判断产品是否到该工位
		IF  fbMachine[1].xTryRun THEN //OR station.xSingleRunning THEN
			station.iStepAuto:= 20;
		ELSE
				IF   station.xEmptyDone THEN
								 xS07MainlineRunPermit:=TRUE;				
								 station.iStepAuto:= 999;
				ELSIF  	arMainlineFixtureData[arCurFixtureNumStation[17]].stProduct.xEmptying  AND 
								arMainlineFixtureData[arCurFixtureNumStation[17]].stProduct.xEmptying  AND 
								NOT  xMainLineSensorReached[1] THEN
 									station.xEmptying:=TRUE;
									station.iStepAuto:= 1000;
				ELSIF NOT  arMainlineFixtureData[arCurFixtureNumStation[17]].xMaterialOnOff AND
							NOT  arMainlineFixtureData[arCurFixtureNumStation[18]].xMaterialOnOff AND  
							NOT  xMainLineSensorReached[1] THEN
								 station.iStepAuto:= 999;
								 xS07MainlineRunPermit:=TRUE;		
				ELSIF	  arMainlineFixtureData[arCurFixtureNumStation[17]].xMaterialOnOff AND    
								arMainlineFixtureData[arCurFixtureNumStation[18]].xMaterialOnOff AND
								xMainLineSensorReached[1]   THEN
								 station.iStepAuto:= 20;
				 END_IF
		END_IF
	20:////Restore_after_Estop_Process1 上载数据流程
			IF  station.xSingleRunning OR fbMachine[1].xTryRun THEN
					station.iStepAuto :=40; 
			ELSIF tsModuleProcess[1].xProcessNotStarted AND NOT  tsModuleProcess[1].xProcessStarted THEN
					station.iStepAuto :=30; (*process not started*)
			ELSIF  tsModuleProcess[1].xProcessStarted AND NOT  tsModuleProcess[1].xProcessCompleted THEN
				 station.iStepAuto := 30;(*process started*)
			ELSIF  tsModuleProcess[1].xProcessCompleted AND NOT tsModuleProcess[1].xQDataCompleted  THEN
					station.iStepAuto :=40 ;(*process completed*)
			ELSIF tsModuleProcess[1].xQDataCompleted THEN
					station.iStepAuto :=40;(*Qdata completed *)
			ELSE
					station.iStepAuto :=21; 
			END_IF	
	21://
				tsModuleProcess[1].xProcessNotStarted:=TRUE;
				station.iStepAuto:= 30;
	30://上载产品数据
				tsModuleProcess[1].xProcessStarted	:=TRUE;
				MEMCPY(ADR(arProcessDataStation[1]),ADR(arMainlineFixtureData[arCurFixtureNumStation[17]]),SIZEOF(arMainlineFixtureData[arCurFixtureNumStation[17]]));
				MEMCPY(ADR(arProcessDataStation[2]),ADR(arMainlineFixtureData[arCurFixtureNumStation[18]]),SIZEOF(arMainlineFixtureData[arCurFixtureNumStation[18]]));
				tsModuleProcess[1].xProcessCompleted	:=TRUE;
				station.iStepAuto:= 40;		
	/////产品流程开始	
	40:	//机械手循环开始  总数为2  最多3
			 	bRobCounter :=1;
				station.iStepAuto:= 50;
	50:////Restore_after_Estop_Process2 /Process3机械手第1/2次取料流程
			IF  station.xSingleRunning OR fbMachine[1].xTryRun THEN
					station.iStepAuto :=60; 
			ELSIF tsModuleProcess[bRobCounter+1].xProcessNotStarted AND NOT  tsModuleProcess[bRobCounter+1].xProcessStarted THEN
					station.iStepAuto :=60; (*process not started*)
			ELSIF  tsModuleProcess[bRobCounter+1].xProcessStarted AND NOT  tsModuleProcess[bRobCounter+1].xProcessCompleted THEN
				 station.iStepAuto := 60;(*process started*)
			ELSIF  tsModuleProcess[bRobCounter+1].xProcessCompleted AND NOT tsModuleProcess[bRobCounter+1].xQDataCompleted  THEN
					station.iStepAuto :=100 ;(*process completed*)
			ELSIF tsModuleProcess[bRobCounter+1].xQDataCompleted THEN
					station.iStepAuto :=100;(*Qdata completed *)
			ELSE
					station.iStepAuto :=60; 
			END_IF
	60://机械手选择取料程序	
			tsModuleProcess[bRobCounter+1].xProcessNotStarted:=TRUE;
			stToRobot1.iMoveMode := CmdRobot1.Cmd_TakePart ;//切换程序
			IF    stFromRobot1.xStepRunning  THEN
			 			stToRobot1.iMoveMode := CmdRobot1.noCmd ;
			 			station.iStepAuto :=70; 
			END_IF
	70://取料子程序运行
			stToRobot1.xStepRunPermit := TRUE ;
			IF stFromRobot1.xStepRunDone THEN
					stToRobot1.xStepRunPermit := FALSE ;
					station.iStepAuto :=80; 
	 		END_IF
	80:	//机械手允许去取料位
				IF  bRobCounter =1 THEN
				 	stToRobot1.xPickPos1Premit :=TRUE;
						IF stFromRobot1.xPickPos1Reached THEN 
							 station.iStepAuto :=85;
						END_IF
				ELSIF bRobCounter =2 THEN
					 stToRobot1.xPickPos2Premit :=TRUE;
					 	IF stFromRobot1.xPickPos2Reached THEN 
							 station.iStepAuto :=85;
						END_IF
				END_IF	
	85://清除信号
				 stToRobot1.xPickPos1Premit := FALSE ;
				 stToRobot1.xPickPos2Premit := FALSE ;	
				  station.iStepAuto :=90;
	90://电动夹爪夹紧
		 tsModuleProcess[bRobCounter+1].xProcessStarted:=TRUE;
		 IF  fbmachine[1].xTryRun THEN 
			 station.iStepAuto :=95;
		 ELSE
			fbClamp.stOper.aClampControl[1]:=TRUE ;
			IF fbClamp.xDone  OR ( fbClamp.xGripClampEmpty AND  fbmachine[1].xTryRun )   THEN
					fbClamp.xExecute :=FALSE ;
					station.iStepAuto :=95;
			END_IF
		END_IF
	95://夹取完成,机械手回中转位
				stToRobot1.xClampPartDone:=TRUE;
			IF   stFromRobot1.xPickTransferPosReached THEN
						 tsModuleProcess[bRobCounter+1].xProcessCompleted:=TRUE;
						station.iStepAuto :=96;
			END_IF
			
	96://复位夹取完成信号
					IF bRobCounter =2 THEN
								xS07MainlineRunPermit:=TRUE;
					END_IF
					stToRobot1.xClampPartDone:=FALSE;
					station.iStepAuto :=97;
	97://等皮带线前进完成后再做放料判断
			IF 	S10_BeltCarrying.station.xDone  AND  NOT station.xDone  AND 
					arBeltLineFixtureData[5].stProduct.xCardLoading_OK   AND
					arBeltLineFixtureData[6].stProduct.xCardLoading_OK THEN
			 	station.iStepAuto :=100;
			END_IF
	100:	////Restore_after_Estop_Process4/Process5 机械手第1/2次放料流程
				station.iStepAuto :=110;
	110://判断该去哪个位置放料
			tsModuleProcess[bRobCounter+3].xProcessNotStarted:=TRUE;
			IF  bRobCounter =1 THEN
			 		IF   arProcessDataStation[1].stProduct.xALL_OK  THEN
					 		IF     NOT S10_BeltCarrying.xBoxSensorReached[1]  AND  NOT S10_BeltCarrying.xBoxSensorReached[2] THEN
					 				iPutPartPosChoose :=stPutPartPosChoose.CardPositon_1;(*卡片1位置 *)
							ELSIF     S10_BeltCarrying.xBoxSensorReached[1]  AND  NOT S10_BeltCarrying.xBoxSensorReached[2] THEN
							 		iPutPartPosChoose :=stPutPartPosChoose.CardPostion_2;(*卡片2位置 *)
							END_IF
					ELSIF  arProcessDataStation[1].stProduct.xPart_NG  THEN
					 		iPutPartPosChoose :=stPutPartPosChoose.NGPositon;(*NG位置*)
					END_IF
					_FirstPosChoose:=iPutPartPosChoose;//记录第一次放置的位置
			ELSIF  bRobCounter =2 THEN
			 		IF   arProcessDataStation[2].stProduct.xALL_OK  THEN 
					 		IF    NOT S10_BeltCarrying.xBoxSensorReached[1]  AND  NOT S10_BeltCarrying.xBoxSensorReached[2] THEN
					 					iPutPartPosChoose :=stPutPartPosChoose.CardPositon_1;(*卡片1位置 *)
							ELSIF  S10_BeltCarrying.xBoxSensorReached[1]   AND  NOT S10_BeltCarrying.xBoxSensorReached[2]  THEN
							 			iPutPartPosChoose :=stPutPartPosChoose.CardPostion_2;(*卡片2位置 *)
							ELSIF	  S10_BeltCarrying.xBoxSensorReached[1]  AND  S10_BeltCarrying.xBoxSensorReached[2] THEN 
							 				iPutPartPosChoose :=stPutPartPosChoose.BufferPostion;(*buffer位置 *)
							END_IF
					ELSIF  arProcessDataStation[2].stProduct.xPart_NG  THEN
					 		iPutPartPosChoose :=stPutPartPosChoose.NGPositon;(*NG位置*)
					END_IF
							_SecondPosChoose:=iPutPartPosChoose;//记录第二次放置位置
			 END_IF
			station.iStepAuto :=111;	
		111://如果第二次和第一次放置的位置相同，请检查程序
					IF		bRobCounter =2 THEN
					 				IF _SecondPosChoose=_FirstPosChoose AND 
										_FirstPosChoose<>stPutPartPosChoose.NGPositon	AND 
										_SecondPosChoose<>stPutPartPosChoose.NGPositon THEN 
										station.iStepAuto :=111;	
									END_IF
					END_IF
						station.iStepAuto :=115;	
		115://检查放料是否被允许
		IF  NOT station.xDone THEN
						IF	S10_BeltCarrying.station.xDone   AND   
									(arBeltLineFixtureData[5].xMaterialOnOff AND 
									arBeltLineFixtureData[6].xMaterialOnOff AND
									arBeltLineFixtureData[5].stProduct.xCardLoading_OK AND
									arBeltLineFixtureData[6].stProduct.xCardLoading_OK ) OR 
									S09_CardCarrying.station.xDisabled  THEN  
									IF   iPutPartPosChoose  =stPutPartPosChoose.CardPositon_1 THEN
												IF  NOT  S10_BeltCarrying.xBoxSensorReached[1] THEN
															station.iStepAuto :=120;    
												ELSE
													station.adwAlarm[1].09	:=	TRUE	;//	S07孔板搬运工位卡片1位置不可重复放置,请检查
												END_IF
									ELSIF	 iPutPartPosChoose  =stPutPartPosChoose.CardPostion_2 THEN
												IF  NOT  S10_BeltCarrying.xBoxSensorReached[2] THEN
															station.iStepAuto :=120;   
												ELSE
														station.adwAlarm[1].10	:=	TRUE	;//	S07孔板搬运工位卡片2位置不可重复放置,请检查 
												END_IF 
									END_IF
							END_IF	
						IF iPutPartPosChoose  =stPutPartPosChoose. BufferPostion THEN 
							 IF  NOT xBufferPosCheckSensor THEN
								 station.iStepAuto :=120;
							 ELSE
									 station.adwAlarm[1].11	:=	TRUE	;//	S07孔板搬运工位Bufffer位置不可重复放置,请检查 
							 END_IF
						ELSIF  iPutPartPosChoose  =stPutPartPosChoose.NGPositon THEN
							 IF  (NOT xNGPosCheckSensor[1] AND NOT  xNGPosCheckSensor[2]) AND   xNGPutBoxPermit  THEN
								 station.iStepAuto :=120;
							 ELSE
								 station.adwAlarm[1].12	:=	TRUE	;//	S07孔板搬运工位NG流道位置不可重复放置,请检查 
							 END_IF	
						END_IF
		END_IF 
	120:	///切换放料程序
			stToRobot1.iMoveMode := CmdRobot1.Cmd_PutPart ;//切换程序
			IF    stFromRobot1.xStepRunning  THEN
			 			stToRobot1.iMoveMode := CmdRobot1.noCmd ;
			 			station.iStepAuto :=125; 
			END_IF
	125://放料子程序运行
			stToRobot1.xStepRunPermit := TRUE ;
			IF stFromRobot1.xStepRunDone THEN
					stToRobot1.xStepRunPermit := FALSE ;
					station.iStepAuto :=130; 
	 		END_IF				
	130:	//机械手开始放料
			IF  fbMachine[1].xTryRun THEN
			 			IF  bRobCounter =1 THEN 
									 stToRobot1.xPutPos1Premit:=TRUE;(*卡片1位置 *)
									 IF stFromRobot1.xPutPos1Reached THEN 
											stToRobot1.xPutPos1Premit := FALSE ;
											station.iStepAuto :=140;
									 END_IF
						ELSIF  	 bRobCounter =2 THEN
											 stToRobot1.xPutPos2Premit:=TRUE;(*卡片2位置 *)
											 IF stFromRobot1.xPutPos2Reached THEN 
													stToRobot1.xPutPos2Premit := FALSE ;
													station.iStepAuto :=140;
											 END_IF
						END_IF
			ELSE
				CASE   iPutPartPosChoose OF
				 	stPutPartPosChoose.CardPositon_1: 
					
										 stToRobot1.xPutPos1Premit:=TRUE;(*卡片1位置 *)
										 IF stFromRobot1.xPutPos1Reached THEN 
												stToRobot1.xPutPos1Premit := FALSE ;
												station.iStepAuto :=140;
										 END_IF
						
					stPutPartPosChoose.CardPostion_2:
							
										 stToRobot1.xPutPos2Premit:=TRUE;(*卡片2位置 *)
										 IF stFromRobot1.xPutPos2Reached THEN 
												stToRobot1.xPutPos2Premit := FALSE ;
												station.iStepAuto :=140;
										 END_IF
					
					stPutPartPosChoose.NGPositon:
				
										stToRobot1.xPutPos3Premit:=TRUE;(*NG流道位置 *)
										IF stFromRobot1.xPutPos3Reached THEN 
											 stToRobot1.xPutPos3Premit := FALSE ;
											 station.iStepAuto :=140;
										END_IF
			
					stPutPartPosChoose.BufferPostion:
					
											stToRobot1.xPutPos4Premit:=TRUE;(*buffer位置 *)
											IF stFromRobot1.xPutPos4Reached THEN 
												 stToRobot1.xPutPos4Premit := FALSE ;
												 station.iStepAuto :=140;
											END_IF
				
					END_CASE
				END_IF
	140://机械手到位，松开夹爪
			tsModuleProcess[bRobCounter+3].xProcessStarted:=TRUE;
			IF fbMachine[1].xTryRun THEN
			 		station.iStepAuto:= 150;
			ELSE
				fbClamp.stOper.aReleaseControl[1]:=TRUE ;
				IF fbClamp.xDone  THEN 
					fbClamp.xExecute :=FALSE ;
					station.iStepAuto:= 150;
				END_IF		
			END_IF
	150://记录放完的位置标志位
		//	IF  iPutPartPosChoose=stPutPartPosChoose.CardPositon_1 THEN
		//	 	xPutBeltLineCompleted[1]:=TRUE;
		//	ELSIF iPutPartPosChoose=stPutPartPosChoose.CardPostion_2 THEN
		//	 	xPutBeltLineCompleted[2]:=TRUE;
		//	END_IF
			station.iStepAuto:= 155;
	155://机械手回中转位置
			tsModuleProcess[bRobCounter+3].xProcessCompleted:=TRUE;
			stToRobot1.xReleasePartDone:=TRUE;
				station.iStepAuto :=156; 
   156://机械手到达中转位置
			 xNGLinePremit:=TRUE;
			IF stFromRobot1.xPickTransferPosReached THEN
			 		stToRobot1.xReleasePartDone:=FALSE;
					station.iStepAuto :=170; 
	 		END_IF	
	170://循环+1
			bRobCounter :=bRobCounter +1;
			station.iStepAuto :=180; 
	180://判断是否继续
			IF   bRobCounter<=2 THEN
				station.iStepAuto :=50; 
			ELSE
				station.iStepAuto :=190; 
			END_IF
	190://是否需要第三次放料	
			IF   	S10_BeltCarrying.xBoxSensorReached[1] AND 
					 NOT S10_BeltCarrying.xBoxSensorReached[2] AND  
					xBufferPosCheckSensor THEN
					station.iStepAuto :=200; 
			ELSE
					station.iStepAuto :=300; 
			END_IF
	200:////Restore_after_Estop_Process6 机械手第三次取料流程
			IF  station.xSingleRunning OR fbMachine[1].xTryRun THEN
					station.iStepAuto :=210; 
			ELSIF tsModuleProcess[6].xProcessNotStarted AND NOT  tsModuleProcess[6].xProcessStarted THEN
					station.iStepAuto :=210; (*process not started*)
			ELSIF  tsModuleProcess[6].xProcessStarted AND NOT  tsModuleProcess[6].xProcessCompleted THEN
				 station.iStepAuto := 210;(*process started*)
			ELSIF  tsModuleProcess[6].xProcessCompleted AND NOT tsModuleProcess[6].xQDataCompleted  THEN
					station.iStepAuto :=260 ;(*process completed*)
			ELSIF tsModuleProcess[6].xQDataCompleted THEN
					station.iStepAuto :=260;(*Qdata completed *)
			ELSE
					station.iStepAuto :=210; 
			END_IF					
	210://	机械手切换到取料程序
			tsModuleProcess[6].xProcessNotStarted:=TRUE;	
			iPickPartPosChoose :=stTakePartPosChoose.BufferPostion; 
			stToRobot1.iMoveMode := CmdRobot1.Cmd_TakePart ;//切换程序
			IF  stFromRobot1.xStepRunning THEN
			 			stToRobot1.iMoveMode := CmdRobot1.noCmd ;
			 			station.iStepAuto :=220; 
			END_IF
	220://取料程序运行
			stToRobot1.xStepRunPermit := TRUE ;
			IF stFromRobot1.xStepRunDone THEN
					stToRobot1.xStepRunPermit := FALSE ;
					station.iStepAuto :=230; 
	 		END_IF	
	230://去Buffer位置的产品
				stToRobot1.xPickPos3Premit := TRUE ;
			 IF stFromRobot1.xPickPos3Reached THEN 
				stToRobot1.xPickPos3Premit := FALSE ;
				station.iStepAuto :=240;
			 END_IF
	240://电动夹爪夹取
			tsModuleProcess[6].xProcessStarted :=TRUE;
			IF NOT fbmachine[1].xTryRun THEN 
				station.iStepAuto :=250;
			ELSE
				fbClamp.stOper.aClampControl[1]:=TRUE ;
				IF fbClamp.xDone  OR ( fbClamp.xGripClampEmpty AND  fbmachine[1].xTryRun )   THEN
						fbClamp.xExecute :=FALSE ;
						station.iStepAuto :=250;
				END_IF
			END_IF
	250://夹取完成
			tsModuleProcess[6].xProcessCompleted:=TRUE; 
			stToRobot1.xClampPartDone :=TRUE;
		IF    stFromRobot1.xPickTransferPosReached THEN
					station.iStepAuto :=260;
		END_IF
	260://机械手切换放料程序
			stToRobot1.iMoveMode := CmdRobot1.Cmd_PutPart ;//切换程序
			IF  stFromRobot1.xStepRunning THEN
			 	stToRobot1.iMoveMode := CmdRobot1.noCmd ;
			 	station.iStepAuto :=265;
			END_IF
	265://运行放料程序
			stToRobot1.xStepRunPermit := TRUE ;
			IF stFromRobot1.xStepRunDone THEN
					stToRobot1.xStepRunPermit := FALSE ;
					station.iStepAuto :=270; 
	 		END_IF	
	270://放到皮带线位置2
			stToRobot1.xPutPos2Premit := TRUE ;
			 IF stFromRobot1.xPutPos4Reached THEN 
				stToRobot1.xPutPos2Premit := FALSE ;
				station.iStepAuto :=280;
			 END_IF				
	280://夹爪松开
			fbClamp.stOper.aReleaseControl[1]:=TRUE ;
			IF fbClamp.xDone  THEN 
			  fbClamp.xExecute :=FALSE ;
			  station.iStepAuto:= 290;
			END_IF		
	290://机械手回参考位置
			stToRobot1.xReleasePartDone:=TRUE;
			IF stFromRobot1.xPickTransferPosReached THEN
					station.iStepAuto :=300; 
	 		END_IF	
	300://清除本地记录
			FOR i:=1 TO gc_ModuleProNo BY 1 DO
				MEMSET(ADR(tsModuleProcess[i]),0,SIZEOF(tsModuleProcess[i]));
			END_FOR
			station.iStepAuto :=999; 
	999://----Single Run Finish----
		IF NOT station.xSingleContinuousRun THEN
			station.xSingleRunFlag:=FALSE;
		END_IF
		station.xCycleEnable:=FALSE;	
		IF arBeltLineFixtureData[5].xMaterialOnOff AND  arBeltLineFixtureData[6].xMaterialOnOff THEN   
					IF  (S10_BeltCarrying.xBoxSensorReached[1] AND S10_BeltCarrying.xBoxSensorReached[2]) THEN 
							station.xDone:=TRUE;
							station.iStepAuto :=0;
					ELSIF 		 NOT  arMainlineFixtureData[arCurFixtureNumStation[17]].xMaterialOnOff AND
										 NOT  arMainlineFixtureData[arCurFixtureNumStation[18]].xMaterialOnOff  THEN///皮带线卡片已到但是主流线产品未到
					 			station.iStepAuto :=0;
					END_IF
		ELSIF   NOT arBeltLineFixtureData[5].xMaterialOnOff AND  NOT arBeltLineFixtureData[6].xMaterialOnOff  THEN
						  station.xDone:=TRUE;
							station.iStepAuto :=0;
		END_IF

{region "清料程序"}
1000://写入数据
	 		 arMainlineFixtureData[arCurFixtureNumStation[17]].xMaterialOnOff:=FALSE;
	 		 arMainlineFixtureData[arCurFixtureNumStation[18]].xMaterialOnOff:=FALSE;
	 		 arMainlineFixtureData[arCurFixtureNumStation[17]].stProduct.xEmptying:=FALSE;
	 		 arMainlineFixtureData[arCurFixtureNumStation[18]].stProduct.xEmptying:=FALSE;
			 station.iStepAuto :=1010;
1010://清料完成
	 	station.xEmptying:=FALSE;
		station.xEmptyDone:=TRUE;
		station.iStepAuto :=0;	
{endregion}
		
		
		
		
		
	ELSE
		;	
END_CASE
(****************NG流道********************)
CASE    iNGStep OF
	0://检查NG流道是否刚放上产品
		IF (xNGPosCheckSensor[1]  OR xNGPosCheckSensor[2]  )AND  xNGLinePremit THEN
				xNGPutBoxPermit:=FALSE;
				xNGLinePremit:=FALSE;
				iNGStep:=iNGStep +1 ;
		END_IF
	1://检查NG满料传感器检测
		arTonDelay[02](IN:= FALSE);
		_AlarmDisable:=FALSE;
		IF  xNGPosCheckSensor[3] THEN
			iNGStep:=iNGStep +1;
		ELSE
			iNGStep:=iNGStep +2 ;
		END_IF
	2:
		IF NOT _AlarmDisable THEN
			station.adwAlarm[1].01:=TRUE;//NG流道满料请处理	
			_AlarmDisable:=TRUE;
		END_IF
		iNGStep:=iNGStep -1 ;
	3://步进JOG速度
				fbAxis[19].rJogVelocity:=10.0;
				iNGStep:=iNGStep +1;
	4://开始JOG到目标位置
			_AlarmDisable:=FALSE;
			arTonDelay[02](IN:=TRUE  , PT:=T#200S , Q=> , ET=> );
			IF   NOT xNGPosCheckSensor[2] AND  NOT xNGPosCheckSensor[1]   THEN
							 fbNGStepMotor.xJogForwardAuto:=FALSE;
							 fbNGStepMotor.xJogForwardHmi:=FALSE;
							 iNGStep:=iNGStep +1;
			ELSE
			 			IF  fbMachine[1].xAutoMode THEN
						   fbNGStepMotor.xJogForwardAuto:=TRUE;
					 ELSIF station.xSingleRunning THEN
							 fbNGStepMotor.xJogForwardHmi:=TRUE;
					 END_IF
			END_IF
			IF  arTonDelay[02].Q  THEN
			 		fbNGStepMotor.xJogForwardAuto:=FALSE;
					fbNGStepMotor.xJogForwardHmi:=FALSE;
					arTonDelay[02](IN:=FALSE);
						iNGStep:=iNGStep +2;
			END_IF
			IF   xNGPosCheckSensor[3] THEN
			 		fbNGStepMotor.xJogForwardAuto:=FALSE;
					fbNGStepMotor.xJogForwardHmi:=FALSE;
						iNGStep:=iNGStep +3;
			END_IF
	5://JOG结束		
						iNGStep:=iNGStep +3;
	6://步进JOG超时，请检查传感器是否正常
		IF   NOT _AlarmDisable THEN
			station.adwAlarm[1].02:=TRUE;//NG流道步进运动超时 ，请检查传感器是否正常
			_AlarmDisable:=TRUE;
		END_IF
		iNGStep:=0;	
	7://NG流道满料 
		IF NOT _AlarmDisable THEN
			station.adwAlarm[1].01:=TRUE;//NG流道满料请处理	
			_AlarmDisable:=TRUE;
		END_IF
		iNGStep:=0;
	8://NG流道动作完成
		xNGPutBoxPermit:=TRUE;
		iNGStep:=0;
END_CASE


END_IF
END_ACTION

ACTION FlowInit:
IF NOT station.xIniting THEN
  station.iStepInit:=0;    
ELSE
//--------------------------------------------初始化步序----------------------------------
CASE station.iStepInit OF	
 0://  
  	IF station.xIniting THEN	
  	  station.iStepInit:=10;	
  	END_IF	
10://复位数据
	stToRobot1.xStepRunPermit :=FALSE ;
	fbClamp.xExecute :=FALSE;
	fbClamp.stOper.xInitControl:=FALSE ;	
	FOR i:=1 TO gc_ModuleProNo BY 1 DO
				MEMSET(ADR(tsModuleProcess[i]),0,SIZEOF(tsModuleProcess[i]));
			END_FOR
	IF  NOT fbMachine[1].xTryRun THEN
		station.iStepInit :=30;
	ELSE
			station.iStepInit :=50;
	 END_IF
	 
